LIN {X 0,Y 318.521,Z 646.616,A -85,B 0,C 180,E1 12916.819,E2 12916.819} C_VEL
LIN {X 0,Y 314.877,Z 667.549,A -85,B 0,C 180,E1 12915.793,E2 12915.793} C_VEL
LIN {X 0,Y 310.481,Z 687.705,A -85,B 0,C 180,E1 12914.459,E2 12914.459} C_VEL
LIN {X 0,Y 305.511,Z 707.389,A -85,B 0,C 180,E1 12912.755,E2 12912.755} C_VEL
LIN {X 0,Y 300.341,Z 725.782,A -85,B 0,C 180,E1 12910.729,E2 12910.729} C_VEL
LIN {X 0,Y 295.179,Z 742.727,A -85,B 0,C 180,E1 12908.414,E2 12908.414} C_VEL
LIN {X 0,Y 290.123,Z 758.694,A -85,B 0,C 180,E1 12905.742,E2 12905.742} C_VEL
LIN {X 0,Y 285.541,Z 773.07,A -85,B 0,C 180,E1 12902.819,E2 12902.819} C_VEL
LIN {X 0,Y 281.238,Z 787.006,A -85,B 0,C 180,E1 12899.38,E2 12899.38} C_VEL
LIN {X 0,Y 277.714,Z 799.537,A -85,B 0,C 180,E1 12895.596,E2 12895.596} C_VEL
LIN {X 0,Y 275.265,Z 809.934,A -85,B 0,C 180,E1 12891.746,E2 12891.746} C_VEL
LIN {X 0,Y 273.777,Z 818.455,A -85,B 0,C 180,E1 12887.864,E2 12887.864} C_VEL
LIN {X 0,Y 273.13,Z 825.558,A -85,B 0,C 180,E1 12883.765,E2 12883.765} C_VEL
LIN {X 0,Y 273.196,Z 830.779,A -85,B 0,C 180,E1 12879.692,E2 12879.692} C_VEL
LIN {X 0,Y 273.612,Z 834.096,A -85,B 0,C 180,E1 12875.873,E2 12875.873} C_VEL
LIN {X 0,Y 273.979,Z 835.824,A -85,B 0,C 180,E1 12872.301,E2 12872.301} C_VEL
LIN {X 0,Y 274.057,Z 836.01,A -85,B 0,C 180,E1 12868.955,E2 12868.955} C_VEL
LIN {X 0,Y 273.763,Z 834.896,A -85,B 0,C 180,E1 12865.391,E2 12865.391} C_VEL
LIN {X 0,Y 273.337,Z 832.235,A -85,B 0,C 180,E1 12861.798,E2 12861.798} C_VEL
LIN {X 0,Y 273.084,Z 827.633,A -85,B 0,C 180,E1 12857.74,E2 12857.74} C_VEL
LIN {X 0,Y 273.452,Z 821.244,A -85,B 0,C 180,E1 12853.648,E2 12853.648} C_VEL
LIN {X 0,Y 274.661,Z 812.965,A -85,B 0,C 180,E1 12849.546,E2 12849.546} C_VEL
LIN {X 0,Y 276.918,Z 802.631,A -85,B 0,C 180,E1 12845.467,E2 12845.467} C_VEL
LIN {X 0,Y 280.149,Z 790.716,A -85,B 0,C 180,E1 12841.662,E2 12841.662} C_VEL
LIN {X 0,Y 284.213,Z 777.257,A -85,B 0,C 180,E1 12838.151,E2 12838.151} C_VEL
LIN {X 0,Y 288.798,Z 762.744,A -85,B 0,C 180,E1 12835.043,E2 12835.043} C_VEL
LIN {X 0,Y 293.673,Z 747.357,A -85,B 0,C 180,E1 12832.329,E2 12832.329} C_VEL
LIN {X 0,Y 298.826,Z 730.575,A -85,B 0,C 180,E1 12829.903,E2 12829.903} C_VEL
LIN {X 0,Y 304.127,Z 712.146,A -85,B 0,C 180,E1 12827.755,E2 12827.755} C_VEL
LIN {X 0,Y 309.042,Z 693.226,A -85,B 0,C 180,E1 12826.004,E2 12826.004} C_VEL
LIN {X 0,Y 313.618,Z 673.067,A -85,B 0,C 180,E1 12824.559,E2 12824.559} C_VEL
LIN {X 0,Y 317.514,Z 652.33,A -85,B 0,C 180,E1 12823.454,E2 12823.454} C_VEL
LIN {X 0,Y 320.333,Z 631.352,A -85,B 0,C 180,E1 12822.639,E2 12822.639} C_VEL
LIN {X 0,Y 322.11,Z 608.021,A -85,B 0,C 180,E1 12822.015,E2 12822.015} C_VEL
LIN {X 0,Y 331.889,Z 436.421,A -85,B 0,C 180,E1 12818.133,E2 12818.133} C_VEL
LIN {X 0,Y 331.118,Z 424.68,A -85,B 0,C 180,E1 12817.587,E2 12817.587} C_VEL
LIN {X 0,Y 322.829,Z 409.225,A -85,B 0,C 180,E1 12815.31,E2 12815.31} C_VEL
LIN {X 0,Y 314.205,Z 394.789,A -85,B 0,C 180,E1 12812.749,E2 12812.749} C_VEL
LIN {X 0,Y 306.355,Z 382.678,A -85,B 0,C 180,E1 12810.173,E2 12810.173} C_VEL
LIN {X 0,Y 298.711,Z 371.628,A -85,B 0,C 180,E1 12807.349,E2 12807.349} C_VEL
LIN {X 0,Y 294.503,Z 363.438,A -85,B 0,C 180,E1 12804.255,E2 12804.255} C_VEL
LIN {X 0,Y 291.847,Z 358.564,A -85,B 0,C 180,E1 12802.139,E2 12802.139} C_VEL
LIN {X 0,Y 289.754,Z 354.487,A -85,B 0,C 180,E1 12800.186,E2 12800.186} C_VEL
LIN {X 0,Y 287.159,Z 349.76,A -85,B 0,C 180,E1 12797.633,E2 12797.633} C_VEL
LIN {X 0,Y 284.83,Z 345.563,A -85,B 0,C 180,E1 12795.056,E2 12795.056} C_VEL
LIN {X 0,Y 281.786,Z 340.679,A -85,B 0,C 180,E1 12791.253,E2 12791.253} C_VEL
LIN {X 0,Y 281.192,Z 339.431,A -85,B 0,C 180,E1 12790.241,E2 12790.241} C_VEL
LIN {X 0,Y 277.823,Z 333.98,A -85,B 0,C 180,E1 12783.507,E2 12783.507} C_VEL
LIN {X 0,Y 276.215,Z 332.418,A -85,B 0,C 180,E1 12777.505,E2 12777.505} C_VEL
LIN {X 0,Y 276.38,Z 332.578,A -85,B 0,C 180,E1 12772.098,E2 12772.098} C_VEL
LIN {X 0,Y 277.952,Z 334.225,A -85,B 0,C 180,E1 12766.901,E2 12766.901} C_VEL
LIN {X 0,Y 281.193,Z 339.671,A -85,B 0,C 180,E1 12760.257,E2 12760.257} C_VEL
LIN {X 0,Y 283.306,Z 343.892,A -85,B 0,C 180,E1 12756.936,E2 12756.936} C_VEL
LIN {X 0,Y 284.176,Z 345.216,A -85,B 0,C 180,E1 12755.911,E2 12755.911} C_VEL
LIN {X 0,Y 286.766,Z 350.132,A -85,B 0,C 180,E1 12752.757,E2 12752.757} C_VEL
LIN {X 0,Y 289.262,Z 355.103,A -85,B 0,C 180,E1 12750.034,E2 12750.034} C_VEL
LIN {X 0,Y 295.268,Z 362.715,A -85,B 0,C 180,E1 12747.366,E2 12747.366} C_VEL
LIN {X 0,Y 303.925,Z 373.809,A -85,B 0,C 180,E1 12744.097,E2 12744.097} C_VEL
LIN {X 0,Y 313.853,Z 387.94,A -85,B 0,C 180,E1 12740.833,E2 12740.833} C_VEL
LIN {X 0,Y 323.057,Z 402.598,A -85,B 0,C 180,E1 12738.136,E2 12738.136} C_VEL
LIN {X 0,Y 331.436,Z 417.301,A -85,B 0,C 180,E1 12735.892,E2 12735.892} C_VEL
LIN {X 0,Y 324.029,Z 570.746,A -85,B 0,C 180,E1 12732.693,E2 12732.693} C_VEL
LIN {X 0,Y 322.622,Z 590.161,A -85,B 0,C 180,E1 12732.013,E2 12732.013} C_VEL
LIN {X 0,Y 320.358,Z 608.777,A -85,B 0,C 180,E1 12731.069,E2 12731.069} C_VEL
LIN {X 0,Y 317.4,Z 626.429,A -85,B 0,C 180,E1 12729.869,E2 12729.869} C_VEL
LIN {X 0,Y 313.615,Z 644.125,A -85,B 0,C 180,E1 12728.322,E2 12728.322} C_VEL
LIN {X 0,Y 309.308,Z 660.695,A -85,B 0,C 180,E1 12726.497,E2 12726.497} C_VEL
LIN {X 0,Y 304.53,Z 676.538,A -85,B 0,C 180,E1 12724.313,E2 12724.313} C_VEL
LIN {X 0,Y 299.564,Z 691.068,A -85,B 0,C 180,E1 12721.826,E2 12721.826} C_VEL
LIN {X 0,Y 294.635,Z 704.227,A -85,B 0,C 180,E1 12719.03,E2 12719.03} C_VEL
LIN {X 0,Y 289.962,Z 715.814,A -85,B 0,C 180,E1 12715.971,E2 12715.971} C_VEL
LIN {X 0,Y 285.729,Z 725.888,A -85,B 0,C 180,E1 12712.638,E2 12712.638} C_VEL
LIN {X 0,Y 282.058,Z 734.454,A -85,B 0,C 180,E1 12709.033,E2 12709.033} C_VEL
LIN {X 0,Y 279.071,Z 741.482,A -85,B 0,C 180,E1 12705.161,E2 12705.161} C_VEL
LIN {X 0,Y 276.972,Z 746.671,A -85,B 0,C 180,E1 12701.241,E2 12701.241} C_VEL
LIN {X 0,Y 275.562,Z 750.342,A -85,B 0,C 180,E1 12697.086,E2 12697.086} C_VEL
LIN {X 0,Y 274.872,Z 752.306,A -85,B 0,C 180,E1 12692.919,E2 12692.919} C_VEL
LIN {X 0,Y 274.762,Z 752.649,A -85,B 0,C 180,E1 12688.749,E2 12688.749} C_VEL
LIN {X 0,Y 275.198,Z 751.384,A -85,B 0,C 180,E1 12684.572,E2 12684.572} C_VEL
LIN {X 0,Y 276.288,Z 748.463,A -85,B 0,C 180,E1 12680.418,E2 12680.418} C_VEL
LIN {X 0,Y 278.158,Z 743.76,A -85,B 0,C 180,E1 12676.277,E2 12676.277} C_VEL
LIN {X 0,Y 280.792,Z 737.489,A -85,B 0,C 180,E1 12672.382,E2 12672.382} C_VEL
LIN {X 0,Y 284.139,Z 729.734,A -85,B 0,C 180,E1 12668.75,E2 12668.75} C_VEL
LIN {X 0,Y 288.037,Z 720.554,A -85,B 0,C 180,E1 12665.384,E2 12665.384} C_VEL
LIN {X 0,Y 292.411,Z 709.978,A -85,B 0,C 180,E1 12662.289,E2 12662.289} C_VEL
LIN {X 0,Y 297.09,Z 698.005,A -85,B 0,C 180,E1 12659.458,E2 12659.458} C_VEL
LIN {X 0,Y 302.111,Z 684.038,A -85,B 0,C 180,E1 12656.789,E2 12656.789} C_VEL
LIN {X 0,Y 307.017,Z 668.867,A -85,B 0,C 180,E1 12654.458,E2 12654.458} C_VEL
LIN {X 0,Y 311.62,Z 652.509,A -85,B 0,C 180,E1 12652.438,E2 12652.438} C_VEL
LIN {X 0,Y 315.588,Z 635.868,A -85,B 0,C 180,E1 12650.799,E2 12650.799} C_VEL
LIN {X 0,Y 318.977,Z 618.266,A -85,B 0,C 180,E1 12649.428,E2 12649.428} C_VEL
LIN {X 0,Y 321.711,Z 599.435,A -85,B 0,C 180,E1 12648.312,E2 12648.312} C_VEL
LIN {X 0,Y 323.578,Z 579.916,A -85,B 0,C 180,E1 12647.482,E2 12647.482} C_VEL
LIN {X 0,Y 324.743,Z 555.923,A -85,B 0,C 180,E1 12646.846,E2 12646.846} C_VEL
LIN {X 0,Y 325.912,Z 530.757,A -85,B 0,C 180,E1 12646.323,E2 12646.323} C_VEL
LIN {X 0,Y 325.604,Z 523.168,A -85,B 0,C 180,E1 12646.04,E2 12646.04} C_VEL
LIN {X 0,Y 322.384,Z 503.34,A -85,B 0,C 180,E1 12644.815,E2 12644.815} C_VEL
LIN {X 0,Y 322.193,Z 496.818,A -85,B 0,C 180,E1 12644.576,E2 12644.576} C_VEL
LIN {X 0,Y 326.056,Z 420.531,A -85,B 0,C 180,E1 12642.97,E2 12642.97} C_VEL
LIN {X 0,Y 317.729,Z 405.913,A -85,B 0,C 180,E1 12640.619,E2 12640.619} C_VEL
LIN {X 0,Y 309.549,Z 392.937,A -85,B 0,C 180,E1 12638.093,E2 12638.093} C_VEL
LIN {X 0,Y 300.513,Z 379.839,A -85,B 0,C 180,E1 12634.968,E2 12634.968} C_VEL
LIN {X 0,Y 291.185,Z 367.626,A -85,B 0,C 180,E1 12631.232,E2 12631.232} C_VEL
LIN {X 0,Y 285.424,Z 360.648,A -85,B 0,C 180,E1 12628.566,E2 12628.566} C_VEL
LIN {X 0,Y 281.908,Z 356.155,A -85,B 0,C 180,E1 12626.651,E2 12626.651} C_VEL
LIN {X 0,Y 279.002,Z 350.696,A -85,B 0,C 180,E1 12622.93,E2 12622.93} C_VEL
LIN {X 0,Y 276.761,Z 346.463,A -85,B 0,C 180,E1 12619.413,E2 12619.413} C_VEL
LIN {X 0,Y 273.571,Z 340.764,A -85,B 0,C 180,E1 12612.025,E2 12612.025} C_VEL
LIN {X 0,Y 272.202,Z 339.441,A -85,B 0,C 180,E1 12606.327,E2 12606.327} C_VEL
LIN {X 0,Y 272.456,Z 339.661,A -85,B 0,C 180,E1 12601.262,E2 12601.262} C_VEL
LIN {X 0,Y 273.881,Z 341.096,A -85,B 0,C 180,E1 12596.442,E2 12596.442} C_VEL
LIN {X 0,Y 277.267,Z 346.64,A -85,B 0,C 180,E1 12589.613,E2 12589.613} C_VEL
LIN {X 0,Y 279.445,Z 350.884,A -85,B 0,C 180,E1 12586.341,E2 12586.341} C_VEL
LIN {X 0,Y 280.36,Z 352.123,A -85,B 0,C 180,E1 12585.333,E2 12585.333} C_VEL
LIN {X 0,Y 282.589,Z 356.255,A -85,B 0,C 180,E1 12582.71,E2 12582.71} C_VEL
LIN {X 0,Y 285.907,Z 362.472,A -85,B 0,C 180,E1 12579.317,E2 12579.317} C_VEL
LIN {X 0,Y 288.869,Z 368.159,A -85,B 0,C 180,E1 12576.76,E2 12576.76} C_VEL
LIN {X 0,Y 290.863,Z 371.534,A -85,B 0,C 180,E1 12575.422,E2 12575.422} C_VEL
LIN {X 0,Y 298.308,Z 382.017,A -85,B 0,C 180,E1 12572.341,E2 12572.341} C_VEL
LIN {X 0,Y 306.047,Z 393.465,A -85,B 0,C 180,E1 12569.523,E2 12569.523} C_VEL
LIN {X 0,Y 314.219,Z 406.761,A -85,B 0,C 180,E1 12566.845,E2 12566.845} C_VEL
LIN {X 0,Y 323.159,Z 422.766,A -85,B 0,C 180,E1 12564.186,E2 12564.186} C_VEL
LIN {X 0,Y 326.324,Z 429.459,A -85,B 0,C 180,E1 12563.27,E2 12563.27} C_VEL
LIN {X 0,Y 326.603,Z 440.209,A -85,B 0,C 180,E1 12562.833,E2 12562.833} C_VEL
LIN {X 0,Y 315.481,Z 623.904,A -85,B 0,C 180,E1 12558.626,E2 12558.626} C_VEL
LIN {X 0,Y 312.841,Z 645.686,A -85,B 0,C 180,E1 12557.856,E2 12557.856} C_VEL
LIN {X 0,Y 309.118,Z 666.476,A -85,B 0,C 180,E1 12556.834,E2 12556.834} C_VEL
LIN {X 0,Y 304.704,Z 686.073,A -85,B 0,C 180,E1 12555.536,E2 12555.536} C_VEL
LIN {X 0,Y 299.76,Z 704.977,A -85,B 0,C 180,E1 12553.907,E2 12553.907} C_VEL
LIN {X 0,Y 294.582,Z 722.809,A -85,B 0,C 180,E1 12551.961,E2 12551.961} C_VEL
LIN {X 0,Y 289.168,Z 739.981,A -85,B 0,C 180,E1 12549.637,E2 12549.637} C_VEL
LIN {X 0,Y 283.936,Z 755.721,A -85,B 0,C 180,E1 12547.024,E2 12547.024} C_VEL
LIN {X 0,Y 278.946,Z 770.642,A -85,B 0,C 180,E1 12543.997,E2 12543.997} C_VEL
LIN {X 0,Y 274.482,Z 784.174,A -85,B 0,C 180,E1 12540.661,E2 12540.661} C_VEL
LIN {X 0,Y 270.765,Z 796.349,A -85,B 0,C 180,E1 12537.013,E2 12537.013} C_VEL
LIN {X 0,Y 267.921,Z 807.109,A -85,B 0,C 180,E1 12533.069,E2 12533.069} C_VEL
LIN {X 0,Y 266.005,Z 816.654,A -85,B 0,C 180,E1 12528.7,E2 12528.7} C_VEL
LIN {X 0,Y 265.206,Z 823.96,A -85,B 0,C 180,E1 12524.408,E2 12524.408} C_VEL
LIN {X 0,Y 265.204,Z 829.303,A -85,B 0,C 180,E1 12520.206,E2 12520.206} C_VEL
LIN {X 0,Y 265.626,Z 832.742,A -85,B 0,C 180,E1 12516.267,E2 12516.267} C_VEL
LIN {X 0,Y 266.028,Z 834.465,A -85,B 0,C 180,E1 12512.8,E2 12512.8} C_VEL
LIN {X 0,Y 266.157,Z 834.862,A -85,B 0,C 180,E1 12509.354,E2 12509.354} C_VEL
LIN {X 0,Y 265.922,Z 834.045,A -85,B 0,C 180,E1 12506.119,E2 12506.119} C_VEL
LIN {X 0,Y 265.435,Z 831.58,A -85,B 0,C 180,E1 12502.206,E2 12502.206} C_VEL
LIN {X 0,Y 265.12,Z 827.563,A -85,B 0,C 180,E1 12498.25,E2 12498.25} C_VEL
LIN {X 0,Y 265.396,Z 821.493,A -85,B 0,C 180,E1 12494.037,E2 12494.037} C_VEL
LIN {X 0,Y 266.529,Z 813.563,A -85,B 0,C 180,E1 12489.811,E2 12489.811} C_VEL
LIN {X 0,Y 268.637,Z 804.049,A -85,B 0,C 180,E1 12485.766,E2 12485.766} C_VEL
LIN {X 0,Y 271.757,Z 792.882,A -85,B 0,C 180,E1 12481.905,E2 12481.905} C_VEL
LIN {X 0,Y 275.768,Z 780.085,A -85,B 0,C 180,E1 12478.284,E2 12478.284} C_VEL
LIN {X 0,Y 280.514,Z 765.839,A -85,B 0,C 180,E1 12474.981,E2 12474.981} C_VEL
LIN {X 0,Y 285.698,Z 750.379,A -85,B 0,C 180,E1 12472.046,E2 12472.046} C_VEL
LIN {X 0,Y 291.038,Z 734.033,A -85,B 0,C 180,E1 12469.512,E2 12469.512} C_VEL
LIN {X 0,Y 296.423,Z 716.509,A -85,B 0,C 180,E1 12467.315,E2 12467.315} C_VEL
LIN {X 0,Y 301.818,Z 697.169,A -85,B 0,C 180,E1 12465.389,E2 12465.389} C_VEL
LIN {X 0,Y 306.581,Z 677.71,A -85,B 0,C 180,E1 12463.885,E2 12463.885} C_VEL
LIN {X 0,Y 310.665,Z 657.913,A -85,B 0,C 180,E1 12462.727,E2 12462.727} C_VEL
LIN {X 0,Y 313.859,Z 637.577,A -85,B 0,C 180,E1 12461.847,E2 12461.847} C_VEL
LIN {X 0,Y 315.922,Z 616.704,A -85,B 0,C 180,E1 12461.203,E2 12461.203} C_VEL
LIN {X 0,Y 326.575,Z 437.654,A -85,B 0,C 180,E1 12457.112,E2 12457.112} C_VEL
LIN {X 0,Y 326.002,Z 428.555,A -85,B 0,C 180,E1 12456.677,E2 12456.677} C_VEL
LIN {X 0,Y 317.855,Z 413.201,A -85,B 0,C 180,E1 12454.323,E2 12454.323} C_VEL
LIN {X 0,Y 308.899,Z 398.062,A -85,B 0,C 180,E1 12451.517,E2 12451.517} C_VEL
LIN {X 0,Y 300.403,Z 384.981,A -85,B 0,C 180,E1 12448.53,E2 12448.53} C_VEL
LIN {X 0,Y 292.847,Z 374.376,A -85,B 0,C 180,E1 12445.534,E2 12445.534} C_VEL
LIN {X 0,Y 290.063,Z 370.213,A -85,B 0,C 180,E1 12444.217,E2 12444.217} C_VEL
LIN {X 0,Y 286.914,Z 364.504,A -85,B 0,C 180,E1 12441.678,E2 12441.678} C_VEL
LIN {X 0,Y 284.984,Z 360.764,A -85,B 0,C 180,E1 12439.896,E2 12439.896} C_VEL
LIN {X 0,Y 282.411,Z 356.076,A -85,B 0,C 180,E1 12437.301,E2 12437.301} C_VEL
LIN {X 0,Y 279.905,Z 351.338,A -85,B 0,C 180,E1 12434.269,E2 12434.269} C_VEL
LIN {X 0,Y 277.516,Z 347.594,A -85,B 0,C 180,E1 12431.218,E2 12431.218} C_VEL
LIN {X 0,Y 276.813,Z 346.091,A -85,B 0,C 180,E1 12429.984,E2 12429.984} C_VEL
LIN {X 0,Y 273.63,Z 340.766,A -85,B 0,C 180,E1 12423.351,E2 12423.351} C_VEL
LIN {X 0,Y 272.02,Z 339.216,A -85,B 0,C 180,E1 12417.261,E2 12417.261} C_VEL
LIN {X 0,Y 272.217,Z 339.429,A -85,B 0,C 180,E1 12411.976,E2 12411.976} C_VEL
LIN {X 0,Y 273.675,Z 341.008,A -85,B 0,C 180,E1 12406.908,E2 12406.908} C_VEL
LIN {X 0,Y 276.735,Z 346.396,A -85,B 0,C 180,E1 12400.365,E2 12400.365} C_VEL
LIN {X 0,Y 278.871,Z 350.546,A -85,B 0,C 180,E1 12396.995,E2 12396.995} C_VEL
LIN {X 0,Y 279.602,Z 351.984,A -85,B 0,C 180,E1 12395.941,E2 12395.941} C_VEL
LIN {X 0,Y 282.03,Z 356.488,A -85,B 0,C 180,E1 12393.012,E2 12393.012} C_VEL
LIN {X 0,Y 285.873,Z 361.055,A -85,B 0,C 180,E1 12391.026,E2 12391.026} C_VEL
LIN {X 0,Y 292.839,Z 369.89,A -85,B 0,C 180,E1 12387.873,E2 12387.873} C_VEL
LIN {X 0,Y 300.999,Z 380.593,A -85,B 0,C 180,E1 12384.69,E2 12384.69} C_VEL
LIN {X 0,Y 310.626,Z 394.567,A -85,B 0,C 180,E1 12381.416,E2 12381.416} C_VEL
LIN {X 0,Y 319.403,Z 408.86,A -85,B 0,C 180,E1 12378.75,E2 12378.75} C_VEL
LIN {X 0,Y 326.078,Z 420.895,A -85,B 0,C 180,E1 12376.879,E2 12376.879} C_VEL
LIN {X 0,Y 318.463,Z 571.358,A -85,B 0,C 180,E1 12373.711,E2 12373.711} C_VEL
LIN {X 0,Y 316.99,Z 590.894,A -85,B 0,C 180,E1 12373.022,E2 12373.022} C_VEL
LIN {X 0,Y 314.593,Z 609.838,A -85,B 0,C 180,E1 12372.052,E2 12372.052} C_VEL
LIN {X 0,Y 311.344,Z 628.339,A -85,B 0,C 180,E1 12370.771,E2 12370.771} C_VEL
LIN {X 0,Y 307.479,Z 645.583,A -85,B 0,C 180,E1 12369.232,E2 12369.232} C_VEL
LIN {X 0,Y 303.009,Z 662.069,A -85,B 0,C 180,E1 12367.383,E2 12367.383} C_VEL
LIN {X 0,Y 298.164,Z 677.501,A -85,B 0,C 180,E1 12365.223,E2 12365.223} C_VEL
LIN {X 0,Y 293.241,Z 691.381,A -85,B 0,C 180,E1 12362.828,E2 12362.828} C_VEL
LIN {X 0,Y 288.068,Z 704.681,A -85,B 0,C 180,E1 12359.987,E2 12359.987} C_VEL
LIN {X 0,Y 283.147,Z 716.394,A -85,B 0,C 180,E1 12356.871,E2 12356.871} C_VEL
LIN {X 0,Y 278.666,Z 726.58,A -85,B 0,C 180,E1 12353.469,E2 12353.469} C_VEL
LIN {X 0,Y 274.765,Z 735.247,A -85,B 0,C 180,E1 12349.78,E2 12349.78} C_VEL
LIN {X 0,Y 271.565,Z 742.37,A -85,B 0,C 180,E1 12345.81,E2 12345.81} C_VEL
LIN {X 0,Y 269.2,Z 747.878,A -85,B 0,C 180,E1 12341.57,E2 12341.57} C_VEL
LIN {X 0,Y 267.705,Z 751.546,A -85,B 0,C 180,E1 12337.295,E2 12337.295} C_VEL
LIN {X 0,Y 266.971,Z 753.508,A -85,B 0,C 180,E1 12333.006,E2 12333.006} C_VEL
LIN {X 0,Y 266.854,Z 753.851,A -85,B 0,C 180,E1 12328.712,E2 12328.712} C_VEL
LIN {X 0,Y 267.317,Z 752.59,A -85,B 0,C 180,E1 12324.419,E2 12324.419} C_VEL
LIN {X 0,Y 268.477,Z 749.667,A -85,B 0,C 180,E1 12320.136,E2 12320.136} C_VEL
LIN {X 0,Y 270.459,Z 744.967,A -85,B 0,C 180,E1 12315.878,E2 12315.878} C_VEL
LIN {X 0,Y 273.239,Z 738.7,A -85,B 0,C 180,E1 12311.879,E2 12311.879} C_VEL
LIN {X 0,Y 276.759,Z 730.951,A -85,B 0,C 180,E1 12308.155,E2 12308.155} C_VEL
LIN {X 0,Y 280.849,Z 721.782,A -85,B 0,C 180,E1 12304.71,E2 12304.71} C_VEL
LIN {X 0,Y 285.424,Z 711.219,A -85,B 0,C 180,E1 12301.549,E2 12301.549} C_VEL
LIN {X 0,Y 290.65,Z 698.387,A -85,B 0,C 180,E1 12298.475,E2 12298.475} C_VEL
LIN {X 0,Y 295.722,Z 684.799,A -85,B 0,C 180,E1 12295.858,E2 12295.858} C_VEL
LIN {X 0,Y 300.837,Z 669.56,A -85,B 0,C 180,E1 12293.494,E2 12293.494} C_VEL
LIN {X 0,Y 305.413,Z 653.91,A -85,B 0,C 180,E1 12291.538,E2 12291.538} C_VEL
LIN {X 0,Y 309.751,Z 636.388,A -85,B 0,C 180,E1 12289.792,E2 12289.792} C_VEL
LIN {X 0,Y 313.272,Z 618.661,A -85,B 0,C 180,E1 12288.406,E2 12288.406} C_VEL
LIN {X 0,Y 316.124,Z 599.539,A -85,B 0,C 180,E1 12287.272,E2 12287.272} C_VEL
LIN {X 0,Y 318.041,Z 579.955,A -85,B 0,C 180,E1 12286.444,E2 12286.444} C_VEL
LIN {X 0,Y 319.275,Z 555.252,A -85,B 0,C 180,E1 12285.793,E2 12285.793} C_VEL
LIN {X 0,Y 322.193,Z 496.818,A -85,B 0,C 180,E1 12284.576,E2 12284.576} C_VEL
LIN {X 0,Y 321.9,Z 489.233,A -85,B 0,C 180,E1 12284.281,E2 12284.281} C_VEL
LIN {X 0,Y 318.898,Z 469.415,A -85,B 0,C 180,E1 12283.022,E2 12283.022} C_VEL
LIN {X 0,Y 318.781,Z 462.892,A -85,B 0,C 180,E1 12282.784,E2 12282.784} C_VEL
LIN {X 0,Y 320.861,Z 424.086,A -85,B 0,C 180,E1 12281.958,E2 12281.958} C_VEL
LIN {X 0,Y 312.608,Z 409.503,A -85,B 0,C 180,E1 12279.501,E2 12279.501} C_VEL
LIN {X 0,Y 303.827,Z 395.623,A -85,B 0,C 180,E1 12276.618,E2 12276.618} C_VEL
LIN {X 0,Y 295.497,Z 383.738,A -85,B 0,C 180,E1 12273.531,E2 12273.531} C_VEL
LIN {X 0,Y 287.709,Z 373.406,A -85,B 0,C 180,E1 12270.202,E2 12270.202} C_VEL
LIN {X 0,Y 282.994,Z 367.663,A -85,B 0,C 180,E1 12267.914,E2 12267.914} C_VEL
LIN {X 0,Y 278.943,Z 362.711,A -85,B 0,C 180,E1 12265.704,E2 12265.704} C_VEL
LIN {X 0,Y 275.103,Z 358.176,A -85,B 0,C 180,E1 12263.339,E2 12263.339} C_VEL
LIN {X 0,Y 274.001,Z 356.757,A -85,B 0,C 180,E1 12262.304,E2 12262.304} C_VEL
LIN {X 0,Y 272.017,Z 352.491,A -85,B 0,C 180,E1 12258.651,E2 12258.651} C_VEL
LIN {X 0,Y 269.226,Z 347.427,A -85,B 0,C 180,E1 12251.787,E2 12251.787} C_VEL
LIN {X 0,Y 268.004,Z 346.218,A -85,B 0,C 180,E1 12245.782,E2 12245.782} C_VEL
LIN {X 0,Y 268.413,Z 346.646,A -85,B 0,C 180,E1 12240.641,E2 12240.641} C_VEL
LIN {X 0,Y 269.761,Z 347.998,A -85,B 0,C 180,E1 12236.388,E2 12236.388} C_VEL
LIN {X 0,Y 272.967,Z 353.552,A -85,B 0,C 180,E1 12229.661,E2 12229.661} C_VEL
LIN {X 0,Y 275.149,Z 357.655,A -85,B 0,C 180,E1 12226.338,E2 12226.338} C_VEL
LIN {X 0,Y 275.934,Z 359.08,A -85,B 0,C 180,E1 12225.307,E2 12225.307} C_VEL
LIN {X 0,Y 278.607,Z 363.943,A -85,B 0,C 180,E1 12222.239,E2 12222.239} C_VEL
LIN {X 0,Y 281.536,Z 369.341,A -85,B 0,C 180,E1 12219.416,E2 12219.416} C_VEL
LIN {X 0,Y 288.409,Z 378.688,A -85,B 0,C 180,E1 12215.962,E2 12215.962} C_VEL
LIN {X 0,Y 295.489,Z 388.867,A -85,B 0,C 180,E1 12212.928,E2 12212.928} C_VEL
LIN {X 0,Y 302.956,Z 400.202,A -85,B 0,C 180,E1 12210.109,E2 12210.109} C_VEL
LIN {X 0,Y 310.665,Z 413.045,A -85,B 0,C 180,E1 12207.488,E2 12207.488} C_VEL
LIN {X 0,Y 319.096,Z 428.488,A -85,B 0,C 180,E1 12204.875,E2 12204.875} C_VEL
LIN {X 0,Y 321.258,Z 433.222,A -85,B 0,C 180,E1 12204.217,E2 12204.217} C_VEL
LIN {X 0,Y 321.382,Z 441.415,A -85,B 0,C 180,E1 12203.892,E2 12203.892} C_VEL
LIN {X 0,Y 309.98,Z 622.999,A -85,B 0,C 180,E1 12199.705,E2 12199.705} C_VEL
LIN {X 0,Y 307.28,Z 644.682,A -85,B 0,C 180,E1 12198.935,E2 12198.935} C_VEL
LIN {X 0,Y 303.47,Z 665.37,A -85,B 0,C 180,E1 12197.916,E2 12197.916} C_VEL
LIN {X 0,Y 298.765,Z 685.59,A -85,B 0,C 180,E1 12196.569,E2 12196.569} C_VEL
LIN {X 0,Y 293.432,Z 705.157,A -85,B 0,C 180,E1 12194.856,E2 12194.856} C_VEL
LIN {X 0,Y 287.796,Z 723.659,A -85,B 0,C 180,E1 12192.78,E2 12192.78} C_VEL
LIN {X 0,Y 282.026,Z 741.029,A -85,B 0,C 180,E1 12190.339,E2 12190.339} C_VEL
LIN {X 0,Y 276.407,Z 757.054,A -85,B 0,C 180,E1 12187.554,E2 12187.554} C_VEL
LIN {X 0,Y 271.431,Z 771.124,A -85,B 0,C 180,E1 12184.56,E2 12184.56} C_VEL
LIN {X 0,Y 266.554,Z 785.146,A -85,B 0,C 180,E1 12180.923,E2 12180.923} C_VEL
LIN {X 0,Y 262.573,Z 797.58,A -85,B 0,C 180,E1 12176.945,E2 12176.945} C_VEL
LIN {X 0,Y 259.636,Z 808.401,A -85,B 0,C 180,E1 12172.649,E2 12172.649} C_VEL
LIN {X 0,Y 257.828,Z 817.539,A -85,B 0,C 180,E1 12168.073,E2 12168.073} C_VEL
LIN {X 0,Y 257.177,Z 824.425,A -85,B 0,C 180,E1 12163.603,E2 12163.603} C_VEL
LIN {X 0,Y 257.326,Z 829.321,A -85,B 0,C 180,E1 12159.275,E2 12159.275} C_VEL
LIN {X 0,Y 257.81,Z 832.213,A -85,B 0,C 180,E1 12155.341,E2 12155.341} C_VEL
LIN {X 0,Y 258.192,Z 833.52,A -85,B 0,C 180,E1 12151.775,E2 12151.775} C_VEL
LIN {X 0,Y 258.221,Z 833.577,A -85,B 0,C 180,E1 12148.669,E2 12148.669} C_VEL
LIN {X 0,Y 257.873,Z 832.472,A -85,B 0,C 180,E1 12145.107,E2 12145.107} C_VEL
LIN {X 0,Y 257.392,Z 829.782,A -85,B 0,C 180,E1 12141.286,E2 12141.286} C_VEL
LIN {X 0,Y 257.157,Z 825.142,A -85,B 0,C 180,E1 12136.967,E2 12136.967} C_VEL
LIN {X 0,Y 257.649,Z 818.824,A -85,B 0,C 180,E1 12132.678,E2 12132.678} C_VEL
LIN {X 0,Y 259.172,Z 810.403,A -85,B 0,C 180,E1 12128.263,E2 12128.263} C_VEL
LIN {X 0,Y 261.847,Z 800.038,A -85,B 0,C 180,E1 12123.953,E2 12123.953} C_VEL
LIN {X 0,Y 265.565,Z 788.098,A -85,B 0,C 180,E1 12119.951,E2 12119.951} C_VEL
LIN {X 0,Y 270.179,Z 774.612,A -85,B 0,C 180,E1 12116.283,E2 12116.283} C_VEL
LIN {X 0,Y 275.675,Z 759.061,A -85,B 0,C 180,E1 12112.852,E2 12112.852} C_VEL
LIN {X 0,Y 281.544,Z 742.29,A -85,B 0,C 180,E1 12109.876,E2 12109.876} C_VEL
LIN {X 0,Y 287.32,Z 724.95,A -85,B 0,C 180,E1 12107.403,E2 12107.403} C_VEL
LIN {X 0,Y 292.908,Z 706.657,A -85,B 0,C 180,E1 12105.318,E2 12105.318} C_VEL
LIN {X 0,Y 298.194,Z 687.393,A -85,B 0,C 180,E1 12103.595,E2 12103.595} C_VEL
LIN {X 0,Y 302.716,Z 668.307,A -85,B 0,C 180,E1 12102.282,E2 12102.282} C_VEL
LIN {X 0,Y 306.579,Z 648.218,A -85,B 0,C 180,E1 12101.243,E2 12101.243} C_VEL
LIN {X 0,Y 309.402,Z 627.413,A -85,B 0,C 180,E1 12100.455,E2 12100.455} C_VEL
LIN {X 0,Y 311.513,Z 598.823,A -85,B 0,C 180,E1 12099.718,E2 12099.718} C_VEL
LIN {X 0,Y 321.355,Z 438.503,A -85,B 0,C 180,E1 12096.039,E2 12096.039} C_VEL
LIN {X 0,Y 320.98,Z 432.39,A -85,B 0,C 180,E1 12095.737,E2 12095.737} C_VEL
LIN {X 0,Y 312.401,Z 416.174,A -85,B 0,C 180,E1 12093.127,E2 12093.127} C_VEL
LIN {X 0,Y 303.613,Z 401.378,A -85,B 0,C 180,E1 12090.201,E2 12090.201} C_VEL
LIN {X 0,Y 295.853,Z 389.496,A -85,B 0,C 180,E1 12087.308,E2 12087.308} C_VEL
LIN {X 0,Y 289.927,Z 380.953,A -85,B 0,C 180,E1 12084.826,E2 12084.826} C_VEL
LIN {X 0,Y 286.251,Z 375.895,A -85,B 0,C 180,E1 12083.138,E2 12083.138} C_VEL
LIN {X 0,Y 281.219,Z 368.69,A -85,B 0,C 180,E1 12080.391,E2 12080.391} C_VEL
LIN {X 0,Y 277.967,Z 362.69,A -85,B 0,C 180,E1 12077.155,E2 12077.155} C_VEL
LIN {X 0,Y 275.164,Z 357.679,A -85,B 0,C 180,E1 12073.876,E2 12073.876} C_VEL
LIN {X 0,Y 272.927,Z 353.563,A -85,B 0,C 180,E1 12070.554,E2 12070.554} C_VEL
LIN {X 0,Y 269.521,Z 347.651,A -85,B 0,C 180,E1 12063.402,E2 12063.402} C_VEL
LIN {X 0,Y 267.908,Z 346.09,A -85,B 0,C 180,E1 12057.433,E2 12057.433} C_VEL
LIN {X 0,Y 268.03,Z 346.237,A -85,B 0,C 180,E1 12052.066,E2 12052.066} C_VEL
LIN {X 0,Y 269.456,Z 347.833,A -85,B 0,C 180,E1 12046.917,E2 12046.917} C_VEL
LIN {X 0,Y 272.292,Z 353.128,A -85,B 0,C 180,E1 12040.478,E2 12040.478} C_VEL
LIN {X 0,Y 274.458,Z 357.249,A -85,B 0,C 180,E1 12036.944,E2 12036.944} C_VEL
LIN {X 0,Y 278.958,Z 362.732,A -85,B 0,C 180,E1 12034.069,E2 12034.069} C_VEL
LIN {X 0,Y 285.034,Z 370.137,A -85,B 0,C 180,E1 12030.869,E2 12030.869} C_VEL
LIN {X 0,Y 291.75,Z 378.69,A -85,B 0,C 180,E1 12027.83,E2 12027.83} C_VEL
LIN {X 0,Y 299.601,Z 389.586,A -85,B 0,C 180,E1 12024.735,E2 12024.735} C_VEL
LIN {X 0,Y 307.927,Z 401.985,A -85,B 0,C 180,E1 12021.847,E2 12021.847} C_VEL
LIN {X 0,Y 317.049,Z 417.21,A -85,B 0,C 180,E1 12019.007,E2 12019.007} C_VEL
LIN {X 0,Y 320.808,Z 424.476,A -85,B 0,C 180,E1 12017.903,E2 12017.903} C_VEL
LIN {X 0,Y 313.005,Z 571.897,A -85,B 0,C 180,E1 12014.768,E2 12014.768} C_VEL
LIN {X 0,Y 311.458,Z 591.638,A -85,B 0,C 180,E1 12014.067,E2 12014.067} C_VEL
LIN {X 0,Y 309.037,Z 610.166,A -85,B 0,C 180,E1 12013.114,E2 12013.114} C_VEL
LIN {X 0,Y 305.73,Z 628.487,A -85,B 0,C 180,E1 12011.847,E2 12011.847} C_VEL
LIN {X 0,Y 301.649,Z 646.164,A -85,B 0,C 180,E1 12010.266,E2 12010.266} C_VEL
LIN {X 0,Y 297.002,Z 662.734,A -85,B 0,C 180,E1 12008.397,E2 12008.397} C_VEL
LIN {X 0,Y 291.753,Z 678.821,A -85,B 0,C 180,E1 12006.117,E2 12006.117} C_VEL
LIN {X 0,Y 286.633,Z 692.662,A -85,B 0,C 180,E1 12003.685,E2 12003.685} C_VEL
LIN {X 0,Y 281.243,Z 705.935,A -85,B 0,C 180,E1 12000.792,E2 12000.792} C_VEL
LIN {X 0,Y 276.104,Z 717.629,A -85,B 0,C 180,E1 11997.614,E2 11997.614} C_VEL
LIN {X 0,Y 271.411,Z 727.804,A -85,B 0,C 180,E1 11994.136,E2 11994.136} C_VEL
LIN {X 0,Y 267.314,Z 736.464,A -85,B 0,C 180,E1 11990.356,E2 11990.356} C_VEL
LIN {X 0,Y 263.941,Z 743.582,A -85,B 0,C 180,E1 11986.279,E2 11986.279} C_VEL
LIN {X 0,Y 261.438,Z 749.087,A -85,B 0,C 180,E1 11981.918,E2 11981.918} C_VEL
LIN {X 0,Y 259.852,Z 752.75,A -85,B 0,C 180,E1 11977.517,E2 11977.517} C_VEL
LIN {X 0,Y 259.071,Z 754.711,A -85,B 0,C 180,E1 11973.097,E2 11973.097} C_VEL
LIN {X 0,Y 258.946,Z 755.052,A -85,B 0,C 180,E1 11968.673,E2 11968.673} C_VEL
LIN {X 0,Y 259.439,Z 753.792,A -85,B 0,C 180,E1 11964.249,E2 11964.249} C_VEL
LIN {X 0,Y 260.673,Z 750.871,A -85,B 0,C 180,E1 11959.838,E2 11959.838} C_VEL
LIN {X 0,Y 262.772,Z 746.174,A -85,B 0,C 180,E1 11955.456,E2 11955.456} C_VEL
LIN {X 0,Y 265.709,Z 739.912,A -85,B 0,C 180,E1 11951.347,E2 11951.347} C_VEL
LIN {X 0,Y 269.412,Z 732.169,A -85,B 0,C 180,E1 11947.527,E2 11947.527} C_VEL
LIN {X 0,Y 273.762,Z 722.884,A -85,B 0,C 180,E1 11943.958,E2 11943.958} C_VEL
LIN {X 0,Y 278.809,Z 711.732,A -85,B 0,C 180,E1 11940.575,E2 11940.575} C_VEL
LIN {X 0,Y 283.938,Z 699.648,A -85,B 0,C 180,E1 11937.64,E2 11937.64} C_VEL
LIN {X 0,Y 289.415,Z 685.558,A -85,B 0,C 180,E1 11934.886,E2 11934.886} C_VEL
LIN {X 0,Y 294.534,Z 670.895,A -85,B 0,C 180,E1 11932.581,E2 11932.581} C_VEL
LIN {X 0,Y 299.506,Z 654.524,A -85,B 0,C 180,E1 11930.51,E2 11930.51} C_VEL
LIN {X 0,Y 303.786,Z 637.887,A -85,B 0,C 180,E1 11928.834,E2 11928.834} C_VEL
LIN {X 0,Y 307.442,Z 620.315,A -85,B 0,C 180,E1 11927.434,E2 11927.434} C_VEL
LIN {X 0,Y 310.382,Z 601.677,A -85,B 0,C 180,E1 11926.301,E2 11926.301} C_VEL
LIN {X 0,Y 312.419,Z 582.429,A -85,B 0,C 180,E1 11925.456,E2 11925.456} C_VEL
LIN {X 0,Y 313.657,Z 560.196,A -85,B 0,C 180,E1 11924.83,E2 11924.83} C_VEL
LIN {X 0,Y 318.781,Z 462.892,A -85,B 0,C 180,E1 11922.784,E2 11922.784} C_VEL
LIN {X 0,Y 318.575,Z 455.305,A -85,B 0,C 180,E1 11922.489,E2 11922.489} C_VEL
LIN {X 0,Y 315.809,Z 435.494,A -85,B 0,C 180,E1 11921.194,E2 11921.194} C_VEL
LIN {X 0,Y 315.722,Z 428.973,A -85,B 0,C 180,E1 11920.948,E2 11920.948} C_VEL
LIN {X 0,Y 315.662,Z 427.477,A -85,B 0,C 180,E1 11920.881,E2 11920.881} C_VEL
LIN {X 0,Y 307.347,Z 412.836,A -85,B 0,C 180,E1 11918.268,E2 11918.268} C_VEL
LIN {X 0,Y 300.149,Z 401.392,A -85,B 0,C 180,E1 11915.777,E2 11915.777} C_VEL
LIN {X 0,Y 292.072,Z 389.55,A -85,B 0,C 180,E1 11912.636,E2 11912.636} C_VEL
LIN {X 0,Y 284.605,Z 379.682,A -85,B 0,C 180,E1 11909.289,E2 11909.289} C_VEL
LIN {X 0,Y 280.969,Z 375.046,A -85,B 0,C 180,E1 11907.442,E2 11907.442} C_VEL
LIN {X 0,Y 277.006,Z 370.123,A -85,B 0,C 180,E1 11905.21,E2 11905.21} C_VEL
LIN {X 0,Y 273.074,Z 365.247,A -85,B 0,C 180,E1 11902.68,E2 11902.68} C_VEL
LIN {X 0,Y 268.53,Z 360.386,A -85,B 0,C 180,E1 11899.241,E2 11899.241} C_VEL
LIN {X 0,Y 267.517,Z 359.038,A -85,B 0,C 180,E1 11898.298,E2 11898.298} C_VEL
LIN {X 0,Y 265.017,Z 354.234,A -85,B 0,C 180,E1 11891.756,E2 11891.756} C_VEL
LIN {X 0,Y 263.83,Z 353.036,A -85,B 0,C 180,E1 11885.655,E2 11885.655} C_VEL
LIN {X 0,Y 264.326,Z 353.564,A -85,B 0,C 180,E1 11880.217,E2 11880.217} C_VEL
LIN {X 0,Y 265.573,Z 354.883,A -85,B 0,C 180,E1 11876.331,E2 11876.331} C_VEL
LIN {X 0,Y 268.502,Z 360.09,A -85,B 0,C 180,E1 11869.921,E2 11869.921} C_VEL
LIN {X 0,Y 270.94,Z 364.479,A -85,B 0,C 180,E1 11866.339,E2 11866.339} C_VEL
LIN {X 0,Y 273.615,Z 369.146,A -85,B 0,C 180,E1 11863.44,E2 11863.44} C_VEL
LIN {X 0,Y 279.467,Z 376.816,A -85,B 0,C 180,E1 11859.858,E2 11859.858} C_VEL
LIN {X 0,Y 286.173,Z 386.133,A -85,B 0,C 180,E1 11856.419,E2 11856.419} C_VEL
LIN {X 0,Y 292.702,Z 395.716,A -85,B 0,C 180,E1 11853.527,E2 11853.527} C_VEL
LIN {X 0,Y 300.012,Z 407.122,A -85,B 0,C 180,E1 11850.666,E2 11850.666} C_VEL
LIN {X 0,Y 307.696,Z 420.322,A -85,B 0,C 180,E1 11847.963,E2 11847.963} C_VEL
LIN {X 0,Y 315.333,Z 434.737,A -85,B 0,C 180,E1 11845.502,E2 11845.502} C_VEL
LIN {X 0,Y 316.291,Z 437.142,A -85,B 0,C 180,E1 11845.188,E2 11845.188} C_VEL
LIN {X 0,Y 316.222,Z 443.384,A -85,B 0,C 180,E1 11844.968,E2 11844.968} C_VEL
LIN {X 0,Y 304.593,Z 622.097,A -85,B 0,C 180,E1 11840.822,E2 11840.822} C_VEL
LIN {X 0,Y 301.813,Z 643.788,A -85,B 0,C 180,E1 11840.049,E2 11840.049} C_VEL
LIN {X 0,Y 297.77,Z 665.007,A -85,B 0,C 180,E1 11838.995,E2 11838.995} C_VEL
LIN {X 0,Y 293.03,Z 684.694,A -85,B 0,C 180,E1 11837.673,E2 11837.673} C_VEL
LIN {X 0,Y 287.673,Z 703.642,A -85,B 0,C 180,E1 11836.009,E2 11836.009} C_VEL
LIN {X 0,Y 282.04,Z 721.457,A -85,B 0,C 180,E1 11834.013,E2 11834.013} C_VEL
LIN {X 0,Y 276.168,Z 738.482,A -85,B 0,C 180,E1 11831.631,E2 11831.631} C_VEL
LIN {X 0,Y 270.255,Z 754.629,A -85,B 0,C 180,E1 11828.835,E2 11828.835} C_VEL
LIN {X 0,Y 264.61,Z 769.797,A -85,B 0,C 180,E1 11825.583,E2 11825.583} C_VEL
LIN {X 0,Y 259.425,Z 783.837,A -85,B 0,C 180,E1 11821.87,E2 11821.87} C_VEL
LIN {X 0,Y 255.163,Z 796.286,A -85,B 0,C 180,E1 11817.794,E2 11817.794} C_VEL
LIN {X 0,Y 251.974,Z 807.122,A -85,B 0,C 180,E1 11813.378,E2 11813.378} C_VEL
LIN {X 0,Y 250.049,Z 815.871,A -85,B 0,C 180,E1 11808.898,E2 11808.898} C_VEL
LIN {X 0,Y 249.253,Z 822.73,A -85,B 0,C 180,E1 11804.401,E2 11804.401} C_VEL
LIN {X 0,Y 249.312,Z 827.793,A -85,B 0,C 180,E1 11799.93,E2 11799.93} C_VEL
LIN {X 0,Y 249.832,Z 830.863,A -85,B 0,C 180,E1 11795.742,E2 11795.742} C_VEL
LIN {X 0,Y 250.258,Z 832.286,A -85,B 0,C 180,E1 11792.061,E2 11792.061} C_VEL
LIN {X 0,Y 250.319,Z 832.404,A -85,B 0,C 180,E1 11788.856,E2 11788.856} C_VEL
LIN {X 0,Y 249.956,Z 831.366,A -85,B 0,C 180,E1 11785.181,E2 11785.181} C_VEL
LIN {X 0,Y 249.439,Z 828.746,A -85,B 0,C 180,E1 11781.239,E2 11781.239} C_VEL
LIN {X 0,Y 249.193,Z 824.191,A -85,B 0,C 180,E1 11776.779,E2 11776.779} C_VEL
LIN {X 0,Y 249.74,Z 817.851,A -85,B 0,C 180,E1 11772.286,E2 11772.286} C_VEL
LIN {X 0,Y 251.355,Z 809.631,A -85,B 0,C 180,E1 11767.797,E2 11767.797} C_VEL
LIN {X 0,Y 254.195,Z 799.352,A -85,B 0,C 180,E1 11763.359,E2 11763.359} C_VEL
LIN {X 0,Y 258.116,Z 787.497,A -85,B 0,C 180,E1 11759.249,E2 11759.249} C_VEL
LIN {X 0,Y 262.962,Z 774.122,A -85,B 0,C 180,E1 11755.492,E2 11755.492} C_VEL
LIN {X 0,Y 268.385,Z 759.548,A -85,B 0,C 180,E1 11752.166,E2 11752.166} C_VEL
LIN {X 0,Y 274.179,Z 743.815,A -85,B 0,C 180,E1 11749.251,E2 11749.251} C_VEL
LIN {X 0,Y 280.09,Z 727.014,A -85,B 0,C 180,E1 11746.735,E2 11746.735} C_VEL
LIN {X 0,Y 285.816,Z 709.369,A -85,B 0,C 180,E1 11744.612,E2 11744.612} C_VEL
LIN {X 0,Y 291.483,Z 689.924,A -85,B 0,C 180,E1 11742.773,E2 11742.773} C_VEL
LIN {X 0,Y 296.536,Z 669.888,A -85,B 0,C 180,E1 11741.326,E2 11741.326} C_VEL
LIN {X 0,Y 300.808,Z 648.932,A -85,B 0,C 180,E1 11740.204,E2 11740.204} C_VEL
LIN {X 0,Y 303.908,Z 627.285,A -85,B 0,C 180,E1 11739.364,E2 11739.364} C_VEL
LIN {X 0,Y 306.061,Z 599.729,A -85,B 0,C 180,E1 11738.64,E2 11738.64} C_VEL
LIN {X 0,Y 316.255,Z 439.472,A -85,B 0,C 180,E1 11734.937,E2 11734.937} C_VEL
LIN {X 0,Y 315.971,Z 436.213,A -85,B 0,C 180,E1 11734.749,E2 11734.749} C_VEL
LIN {X 0,Y 308.414,Z 421.704,A -85,B 0,C 180,E1 11732.338,E2 11732.338} C_VEL
LIN {X 0,Y 300.211,Z 407.543,A -85,B 0,C 180,E1 11729.477,E2 11729.477} C_VEL
LIN {X 0,Y 292.84,Z 396.03,A -85,B 0,C 180,E1 11726.624,E2 11726.624} C_VEL
LIN {X 0,Y 287.054,Z 387.519,A -85,B 0,C 180,E1 11724.104,E2 11724.104} C_VEL
LIN {X 0,Y 283.294,Z 382.254,A -85,B 0,C 180,E1 11722.297,E2 11722.297} C_VEL
LIN {X 0,Y 277.653,Z 374.456,A -85,B 0,C 180,E1 11719.238,E2 11719.238} C_VEL
LIN {X 0,Y 273.404,Z 368.944,A -85,B 0,C 180,E1 11716.573,E2 11716.573} C_VEL
LIN {X 0,Y 270.804,Z 364.328,A -85,B 0,C 180,E1 11713.668,E2 11713.668} C_VEL
LIN {X 0,Y 268.482,Z 360.116,A -85,B 0,C 180,E1 11710.297,E2 11710.297} C_VEL
LIN {X 0,Y 265.269,Z 354.401,A -85,B 0,C 180,E1 11703.241,E2 11703.241} C_VEL
LIN {X 0,Y 263.711,Z 352.868,A -85,B 0,C 180,E1 11696.957,E2 11696.957} C_VEL
LIN {X 0,Y 263.979,Z 353.221,A -85,B 0,C 180,E1 11691.285,E2 11691.285} C_VEL
LIN {X 0,Y 265.225,Z 354.68,A -85,B 0,C 180,E1 11686.927,E2 11686.927} C_VEL
LIN {X 0,Y 267.657,Z 359.152,A -85,B 0,C 180,E1 11681.26,E2 11681.26} C_VEL
LIN {X 0,Y 272.055,Z 364.369,A -85,B 0,C 180,E1 11677.756,E2 11677.756} C_VEL
LIN {X 0,Y 273.384,Z 365.807,A -85,B 0,C 180,E1 11676.848,E2 11676.848} C_VEL
LIN {X 0,Y 277.358,Z 370.442,A -85,B 0,C 180,E1 11674.367,E2 11674.367} C_VEL
LIN {X 0,Y 282.945,Z 377.568,A -85,B 0,C 180,E1 11671.333,E2 11671.333} C_VEL
LIN {X 0,Y 289.194,Z 385.686,A -85,B 0,C 180,E1 11668.412,E2 11668.412} C_VEL
LIN {X 0,Y 296.958,Z 396.688,A -85,B 0,C 180,E1 11665.251,E2 11665.251} C_VEL
LIN {X 0,Y 305.116,Z 409.234,A -85,B 0,C 180,E1 11662.326,E2 11662.326} C_VEL
LIN {X 0,Y 313.511,Z 423.635,A -85,B 0,C 180,E1 11659.623,E2 11659.623} C_VEL
LIN {X 0,Y 315.646,Z 427.98,A -85,B 0,C 180,E1 11658.962,E2 11658.962} C_VEL
LIN {X 0,Y 307.654,Z 572.466,A -85,B 0,C 180,E1 11655.861,E2 11655.861} C_VEL
LIN {X 0,Y 306.034,Z 592.378,A -85,B 0,C 180,E1 11655.15,E2 11655.15} C_VEL
LIN {X 0,Y 303.473,Z 611.223,A -85,B 0,C 180,E1 11654.172,E2 11654.172} C_VEL
LIN {X 0,Y 299.921,Z 630.065,A -85,B 0,C 180,E1 11652.849,E2 11652.849} C_VEL
LIN {X 0,Y 295.686,Z 647.616,A -85,B 0,C 180,E1 11651.252,E2 11651.252} C_VEL
LIN {X 0,Y 290.843,Z 664.176,A -85,B 0,C 180,E1 11649.352,E2 11649.352} C_VEL
LIN {X 0,Y 285.626,Z 679.555,A -85,B 0,C 180,E1 11647.145,E2 11647.145} C_VEL
LIN {X 0,Y 280.092,Z 693.944,A -85,B 0,C 180,E1 11644.581,E2 11644.581} C_VEL
LIN {X 0,Y 274.476,Z 707.191,A -85,B 0,C 180,E1 11641.638,E2 11641.638} C_VEL
LIN {X 0,Y 269.11,Z 718.867,A -85,B 0,C 180,E1 11638.396,E2 11638.396} C_VEL
LIN {X 0,Y 264.194,Z 729.029,A -85,B 0,C 180,E1 11634.839,E2 11634.839} C_VEL
LIN {X 0,Y 259.891,Z 737.68,A -85,B 0,C 180,E1 11630.964,E2 11630.964} C_VEL
LIN {X 0,Y 256.336,Z 744.792,A -85,B 0,C 180,E1 11626.776,E2 11626.776} C_VEL
LIN {X 0,Y 253.686,Z 750.293,A -85,B 0,C 180,E1 11622.288,E2 11622.288} C_VEL
LIN {X 0,Y 252.003,Z 753.954,A -85,B 0,C 180,E1 11617.753,E2 11617.753} C_VEL
LIN {X 0,Y 251.171,Z 755.913,A -85,B 0,C 180,E1 11613.195,E2 11613.195} C_VEL
LIN {X 0,Y 251.039,Z 756.254,A -85,B 0,C 180,E1 11608.631,E2 11608.631} C_VEL
LIN {X 0,Y 251.564,Z 754.995,A -85,B 0,C 180,E1 11604.069,E2 11604.069} C_VEL
LIN {X 0,Y 252.876,Z 752.076,A -85,B 0,C 180,E1 11599.521,E2 11599.521} C_VEL
LIN {X 0,Y 255.102,Z 747.382,A -85,B 0,C 180,E1 11595.009,E2 11595.009} C_VEL
LIN {X 0,Y 258.204,Z 741.123,A -85,B 0,C 180,E1 11590.783,E2 11590.783} C_VEL
LIN {X 0,Y 262.173,Z 733.239,A -85,B 0,C 180,E1 11586.798,E2 11586.798} C_VEL
LIN {X 0,Y 266.893,Z 723.638,A -85,B 0,C 180,E1 11583.045,E2 11583.045} C_VEL
LIN {X 0,Y 271.94,Z 712.971,A -85,B 0,C 180,E1 11579.755,E2 11579.755} C_VEL
LIN {X 0,Y 277.289,Z 700.908,A -85,B 0,C 180,E1 11576.765,E2 11576.765} C_VEL
LIN {X 0,Y 282.99,Z 686.848,A -85,B 0,C 180,E1 11573.966,E2 11573.966} C_VEL
LIN {X 0,Y 288.434,Z 671.864,A -85,B 0,C 180,E1 11571.577,E2 11571.577} C_VEL
LIN {X 0,Y 293.469,Z 655.921,A -85,B 0,C 180,E1 11569.532,E2 11569.532} C_VEL
LIN {X 0,Y 298.059,Z 638.753,A -85,B 0,C 180,E1 11567.781,E2 11567.781} C_VEL
LIN {X 0,Y 301.939,Z 620.702,A -85,B 0,C 180,E1 11566.337,E2 11566.337} C_VEL
LIN {X 0,Y 305.048,Z 601.447,A -85,B 0,C 180,E1 11565.171,E2 11565.171} C_VEL
LIN {X 0,Y 307.146,Z 581.799,A -85,B 0,C 180,E1 11564.321,E2 11564.321} C_VEL
LIN {X 0,Y 308.502,Z 557.357,A -85,B 0,C 180,E1 11563.657,E2 11563.657} C_VEL
LIN {X 0,Y 315.722,Z 428.973,A -85,B 0,C 180,E1 11560.948,E2 11560.948} C_VEL
LIN {X 0,Y 315.453,Z 426.101,A -85,B 0,C 180,E1 11560.784,E2 11560.784} C_VEL
LIN {X 0,Y 314.164,Z 422.942,A -85,B 0,C 180,E1 11560.365,E2 11560.365} C_VEL
LIN {X 0,Y 311.128,Z 419.574,A -85,B 0,C 180,E1 11559.498,E2 11559.498} C_VEL
LIN {X 0,Y 301.539,Z 414.029,A -85,B 0,C 180,E1 11556.707,E2 11556.707} C_VEL
LIN {X 0,Y 299.386,Z 411.597,A -85,B 0,C 180,E1 11555.977,E2 11555.977} C_VEL
LIN {X 0,Y 291.54,Z 399.548,A -85,B 0,C 180,E1 11552.929,E2 11552.929} C_VEL
LIN {X 0,Y 283.395,Z 388.069,A -85,B 0,C 180,E1 11549.252,E2 11549.252} C_VEL
LIN {X 0,Y 278.605,Z 382.043,A -85,B 0,C 180,E1 11546.77,E2 11546.77} C_VEL
LIN {X 0,Y 274.918,Z 377.366,A -85,B 0,C 180,E1 11544.604,E2 11544.604} C_VEL
LIN {X 0,Y 270.738,Z 372.222,A -85,B 0,C 180,E1 11541.787,E2 11541.787} C_VEL
LIN {X 0,Y 266.769,Z 367.583,A -85,B 0,C 180,E1 11538.578,E2 11538.578} C_VEL
LIN {X 0,Y 260.852,Z 361.011,A -85,B 0,C 180,E1 11531.498,E2 11531.498} C_VEL
LIN {X 0,Y 259.657,Z 359.856,A -85,B 0,C 180,E1 11525.525,E2 11525.525} C_VEL
LIN {X 0,Y 260.201,Z 360.429,A -85,B 0,C 180,E1 11520,E2 11520} C_VEL
LIN {X 0,Y 261.322,Z 361.624,A -85,B 0,C 180,E1 11516.491,E2 11516.491} C_VEL
LIN {X 0,Y 264.546,Z 367.06,A -85,B 0,C 180,E1 11510.098,E2 11510.098} C_VEL
LIN {X 0,Y 268.091,Z 371.757,A -85,B 0,C 180,E1 11506.751,E2 11506.751} C_VEL
LIN {X 0,Y 273.021,Z 378.307,A -85,B 0,C 180,E1 11503.074,E2 11503.074} C_VEL
LIN {X 0,Y 277.486,Z 384.308,A -85,B 0,C 180,E1 11500.312,E2 11500.312} C_VEL
LIN {X 0,Y 283.769,Z 393.268,A -85,B 0,C 180,E1 11496.977,E2 11496.977} C_VEL
LIN {X 0,Y 289.947,Z 402.565,A -85,B 0,C 180,E1 11494.137,E2 11494.137} C_VEL
LIN {X 0,Y 297.098,Z 414.031,A -85,B 0,C 180,E1 11491.233,E2 11491.233} C_VEL
LIN {X 0,Y 305.535,Z 428.951,A -85,B 0,C 180,E1 11488.179,E2 11488.179} C_VEL
LIN {X 0,Y 311.41,Z 440.745,A -85,B 0,C 180,E1 11486.205,E2 11486.205} C_VEL
LIN {X 0,Y 299.939,Z 613.756,A -85,B 0,C 180,E1 11482.177,E2 11482.177} C_VEL
LIN {X 0,Y 297.737,Z 634.349,A -85,B 0,C 180,E1 11481.537,E2 11481.537} C_VEL
LIN {X 0,Y 294.375,Z 654.325,A -85,B 0,C 180,E1 11480.673,E2 11480.673} C_VEL
LIN {X 0,Y 289.873,Z 674.284,A -85,B 0,C 180,E1 11479.512,E2 11479.512} C_VEL
LIN {X 0,Y 284.573,Z 693.791,A -85,B 0,C 180,E1 11477.995,E2 11477.995} C_VEL
LIN {X 0,Y 278.62,Z 712.855,A -85,B 0,C 180,E1 11476.067,E2 11476.067} C_VEL
LIN {X 0,Y 272.428,Z 730.666,A -85,B 0,C 180,E1 11473.773,E2 11473.773} C_VEL
LIN {X 0,Y 266.189,Z 747.277,A -85,B 0,C 180,E1 11471.095,E2 11471.095} C_VEL
LIN {X 0,Y 260.188,Z 762.629,A -85,B 0,C 180,E1 11468.022,E2 11468.022} C_VEL
LIN {X 0,Y 254.823,Z 776.222,A -85,B 0,C 180,E1 11464.675,E2 11464.675} C_VEL
LIN {X 0,Y 249.934,Z 789.048,A -85,B 0,C 180,E1 11460.8,E2 11460.8} C_VEL
LIN {X 0,Y 245.999,Z 800.41,A -85,B 0,C 180,E1 11456.556,E2 11456.556} C_VEL
LIN {X 0,Y 243.195,Z 810.243,A -85,B 0,C 180,E1 11451.97,E2 11451.97} C_VEL
LIN {X 0,Y 241.661,Z 818.097,A -85,B 0,C 180,E1 11447.331,E2 11447.331} C_VEL
LIN {X 0,Y 241.215,Z 824.117,A -85,B 0,C 180,E1 11442.69,E2 11442.69} C_VEL
LIN {X 0,Y 241.538,Z 828.112,A -85,B 0,C 180,E1 11438.33,E2 11438.33} C_VEL
LIN {X 0,Y 242.114,Z 830.426,A -85,B 0,C 180,E1 11434.263,E2 11434.263} C_VEL
LIN {X 0,Y 242.425,Z 831.259,A -85,B 0,C 180,E1 11430.709,E2 11430.709} C_VEL
LIN {X 0,Y 242.269,Z 830.908,A -85,B 0,C 180,E1 11427.123,E2 11427.123} C_VEL
LIN {X 0,Y 241.766,Z 829.214,A -85,B 0,C 180,E1 11423.35,E2 11423.35} C_VEL
LIN {X 0,Y 241.279,Z 825.816,A -85,B 0,C 180,E1 11419.011,E2 11419.011} C_VEL
LIN {X 0,Y 241.392,Z 820.517,A -85,B 0,C 180,E1 11414.382,E2 11414.382} C_VEL
LIN {X 0,Y 242.576,Z 812.939,A -85,B 0,C 180,E1 11409.491,E2 11409.491} C_VEL
LIN {X 0,Y 244.961,Z 803.735,A -85,B 0,C 180,E1 11404.882,E2 11404.882} C_VEL
LIN {X 0,Y 248.487,Z 793.032,A -85,B 0,C 180,E1 11400.601,E2 11400.601} C_VEL
LIN {X 0,Y 252.959,Z 780.921,A -85,B 0,C 180,E1 11396.674,E2 11396.674} C_VEL
LIN {X 0,Y 258.222,Z 767.453,A -85,B 0,C 180,E1 11393.119,E2 11393.119} C_VEL
LIN {X 0,Y 264.176,Z 752.263,A -85,B 0,C 180,E1 11389.865,E2 11389.865} C_VEL
LIN {X 0,Y 270.488,Z 735.645,A -85,B 0,C 180,E1 11387.001,E2 11387.001} C_VEL
LIN {X 0,Y 276.674,Z 718.278,A -85,B 0,C 180,E1 11384.61,E2 11384.61} C_VEL
LIN {X 0,Y 282.584,Z 700.006,A -85,B 0,C 180,E1 11382.613,E2 11382.613} C_VEL
LIN {X 0,Y 287.937,Z 681.319,A -85,B 0,C 180,E1 11381.018,E2 11381.018} C_VEL
LIN {X 0,Y 292.634,Z 662.062,A -85,B 0,C 180,E1 11379.758,E2 11379.758} C_VEL
LIN {X 0,Y 296.561,Z 641.568,A -85,B 0,C 180,E1 11378.763,E2 11378.763} C_VEL
LIN {X 0,Y 299.288,Z 620.33,A -85,B 0,C 180,E1 11378.017,E2 11378.017} C_VEL
LIN {X 0,Y 311.297,Z 441.152,A -85,B 0,C 180,E1 11373.832,E2 11373.832} C_VEL
LIN {X 0,Y 310.816,Z 439.448,A -85,B 0,C 180,E1 11373.649,E2 11373.649} C_VEL
LIN {X 0,Y 302.479,Z 423.487,A -85,B 0,C 180,E1 11370.821,E2 11370.821} C_VEL
LIN {X 0,Y 294.957,Z 410.543,A -85,B 0,C 180,E1 11368.001,E2 11368.001} C_VEL
LIN {X 0,Y 287.632,Z 398.981,A -85,B 0,C 180,E1 11364.928,E2 11364.928} C_VEL
LIN {X 0,Y 281.321,Z 389.864,A -85,B 0,C 180,E1 11361.912,E2 11361.912} C_VEL
LIN {X 0,Y 275.621,Z 381.795,A -85,B 0,C 180,E1 11358.726,E2 11358.726} C_VEL
LIN {X 0,Y 271.339,Z 376.126,A -85,B 0,C 180,E1 11355.933,E2 11355.933} C_VEL
LIN {X 0,Y 267.869,Z 371.581,A -85,B 0,C 180,E1 11353.271,E2 11353.271} C_VEL
LIN {X 0,Y 264.423,Z 366.898,A -85,B 0,C 180,E1 11350.016,E2 11350.016} C_VEL
LIN {X 0,Y 261.036,Z 361.164,A -85,B 0,C 180,E1 11343.073,E2 11343.073} C_VEL
LIN {X 0,Y 259.523,Z 359.666,A -85,B 0,C 180,E1 11336.687,E2 11336.687} C_VEL
LIN {X 0,Y 259.871,Z 360.112,A -85,B 0,C 180,E1 11330.923,E2 11330.923} C_VEL
LIN {X 0,Y 261.203,Z 361.397,A -85,B 0,C 180,E1 11327.397,E2 11327.397} C_VEL
LIN {X 0,Y 265.33,Z 366.168,A -85,B 0,C 180,E1 11322.433,E2 11322.433} C_VEL
LIN {X 0,Y 266.687,Z 367.503,A -85,B 0,C 180,E1 11321.19,E2 11321.19} C_VEL
LIN {X 0,Y 270.552,Z 372.073,A -85,B 0,C 180,E1 11318.083,E2 11318.083} C_VEL
LIN {X 0,Y 271.984,Z 373.859,A -85,B 0,C 180,E1 11317.065,E2 11317.065} C_VEL
LIN {X 0,Y 276.235,Z 379.016,A -85,B 0,C 180,E1 11314.371,E2 11314.371} C_VEL
LIN {X 0,Y 280.703,Z 384.74,A -85,B 0,C 180,E1 11311.896,E2 11311.896} C_VEL
LIN {X 0,Y 286.718,Z 392.744,A -85,B 0,C 180,E1 11308.986,E2 11308.986} C_VEL
LIN {X 0,Y 294.761,Z 404.38,A -85,B 0,C 180,E1 11305.612,E2 11305.612} C_VEL
LIN {X 0,Y 303.115,Z 417.764,A -85,B 0,C 180,E1 11302.541,E2 11302.541} C_VEL
LIN {X 0,Y 310.604,Z 431.188,A -85,B 0,C 180,E1 11300.064,E2 11300.064} C_VEL
LIN {X 0,Y 302.407,Z 573.246,A -85,B 0,C 180,E1 11296.987,E2 11296.987} C_VEL
LIN {X 0,Y 300.706,Z 593.258,A -85,B 0,C 180,E1 11296.265,E2 11296.265} C_VEL
LIN {X 0,Y 298.016,Z 612.277,A -85,B 0,C 180,E1 11295.268,E2 11295.268} C_VEL
LIN {X 0,Y 294.452,Z 630.537,A -85,B 0,C 180,E1 11293.979,E2 11293.979} C_VEL
LIN {X 0,Y 290.057,Z 648.192,A -85,B 0,C 180,E1 11292.368,E2 11292.368} C_VEL
LIN {X 0,Y 284.883,Z 665.271,A -85,B 0,C 180,E1 11290.393,E2 11290.393} C_VEL
LIN {X 0,Y 279.376,Z 680.87,A -85,B 0,C 180,E1 11288.122,E2 11288.122} C_VEL
LIN {X 0,Y 273.622,Z 695.221,A -85,B 0,C 180,E1 11285.521,E2 11285.521} C_VEL
LIN {X 0,Y 267.772,Z 708.444,A -85,B 0,C 180,E1 11282.526,E2 11282.526} C_VEL
LIN {X 0,Y 262.169,Z 720.104,A -85,B 0,C 180,E1 11279.219,E2 11279.219} C_VEL
LIN {X 0,Y 257.021,Z 730.255,A -85,B 0,C 180,E1 11275.582,E2 11275.582} C_VEL
LIN {X 0,Y 252.501,Z 738.898,A -85,B 0,C 180,E1 11271.608,E2 11271.608} C_VEL
LIN {X 0,Y 248.751,Z 746.004,A -85,B 0,C 180,E1 11267.304,E2 11267.304} C_VEL
LIN {X 0,Y 245.944,Z 751.501,A -85,B 0,C 180,E1 11262.681,E2 11262.681} C_VEL
LIN {X 0,Y 244.158,Z 755.158,A -85,B 0,C 180,E1 11258.003,E2 11258.003} C_VEL
LIN {X 0,Y 243.272,Z 757.115,A -85,B 0,C 180,E1 11253.299,E2 11253.299} C_VEL
LIN {X 0,Y 243.132,Z 757.455,A -85,B 0,C 180,E1 11248.586,E2 11248.586} C_VEL
LIN {X 0,Y 243.691,Z 756.197,A -85,B 0,C 180,E1 11243.876,E2 11243.876} C_VEL
LIN {X 0,Y 245.087,Z 753.28,A -85,B 0,C 180,E1 11239.184,E2 11239.184} C_VEL
LIN {X 0,Y 247.447,Z 748.588,A -85,B 0,C 180,E1 11234.533,E2 11234.533} C_VEL
LIN {X 0,Y 250.725,Z 742.333,A -85,B 0,C 180,E1 11230.187,E2 11230.187} C_VEL
LIN {X 0,Y 255.002,Z 734.264,A -85,B 0,C 180,E1 11226.008,E2 11226.008} C_VEL
LIN {X 0,Y 259.856,Z 724.856,A -85,B 0,C 180,E1 11222.25,E2 11222.25} C_VEL
LIN {X 0,Y 265.196,Z 714.075,A -85,B 0,C 180,E1 11218.855,E2 11218.855} C_VEL
LIN {X 0,Y 270.812,Z 701.935,A -85,B 0,C 180,E1 11215.795,E2 11215.795} C_VEL
LIN {X 0,Y 276.596,Z 688.252,A -85,B 0,C 180,E1 11213.025,E2 11213.025} C_VEL
LIN {X 0,Y 282.168,Z 673.561,A -85,B 0,C 180,E1 11210.634,E2 11210.634} C_VEL
LIN {X 0,Y 287.521,Z 657.318,A -85,B 0,C 180,E1 11208.513,E2 11208.513} C_VEL
LIN {X 0,Y 292.369,Z 639.895,A -85,B 0,C 180,E1 11206.712,E2 11206.712} C_VEL
LIN {X 0,Y 296.306,Z 622.353,A -85,B 0,C 180,E1 11205.288,E2 11205.288} C_VEL
LIN {X 0,Y 299.493,Z 603.691,A -85,B 0,C 180,E1 11204.131,E2 11204.131} C_VEL
LIN {X 0,Y 301.707,Z 584.601,A -85,B 0,C 180,E1 11203.27,E2 11203.27} C_VEL
LIN {X 0,Y 303.053,Z 563.144,A -85,B 0,C 180,E1 11202.641,E2 11202.641} C_VEL
LIN {X 0,Y 310.65,Z 431.116,A -85,B 0,C 180,E1 11199.8,E2 11199.8} C_VEL
LIN {X 0,Y 302.651,Z 416.894,A -85,B 0,C 180,E1 11197.139,E2 11197.139} C_VEL
LIN {X 0,Y 299.386,Z 411.597,A -85,B 0,C 180,E1 11195.977,E2 11195.977} C_VEL
LIN {X 0,Y 296.103,Z 407.989,A -85,B 0,C 180,E1 11194.815,E2 11194.815} C_VEL
LIN {X 0,Y 288.445,Z 403.386,A -85,B 0,C 180,E1 11192.017,E2 11192.017} C_VEL
LIN {X 0,Y 284.803,Z 400.362,A -85,B 0,C 180,E1 11190.49,E2 11190.49} C_VEL
LIN {X 0,Y 284.011,Z 399.335,A -85,B 0,C 180,E1 11190.122,E2 11190.122} C_VEL
LIN {X 0,Y 277.331,Z 390.187,A -85,B 0,C 180,E1 11186.671,E2 11186.671} C_VEL
LIN {X 0,Y 273.037,Z 384.773,A -85,B 0,C 180,E1 11184.099,E2 11184.099} C_VEL
LIN {X 0,Y 268.964,Z 379.69,A -85,B 0,C 180,E1 11181.251,E2 11181.251} C_VEL
LIN {X 0,Y 264.482,Z 374.303,A -85,B 0,C 180,E1 11177.377,E2 11177.377} C_VEL
LIN {X 0,Y 259.636,Z 368.814,A -85,B 0,C 180,E1 11171.102,E2 11171.102} C_VEL
LIN {X 0,Y 257.497,Z 367.549,A -85,B 0,C 180,E1 11164.901,E2 11164.901} C_VEL
LIN {X 0,Y 258.026,Z 368.268,A -85,B 0,C 180,E1 11159.112,E2 11159.112} C_VEL
LIN {X 0,Y 259.052,Z 369.438,A -85,B 0,C 180,E1 11156.46,E2 11156.46} C_VEL
LIN {X 0,Y 263.131,Z 374.76,A -85,B 0,C 180,E1 11150.486,E2 11150.486} C_VEL
LIN {X 0,Y 266.716,Z 379.556,A -85,B 0,C 180,E1 11147.002,E2 11147.002} C_VEL
LIN {X 0,Y 271.243,Z 385.883,A -85,B 0,C 180,E1 11143.511,E2 11143.511} C_VEL
LIN {X 0,Y 275.28,Z 391.416,A -85,B 0,C 180,E1 11140.92,E2 11140.92} C_VEL
LIN {X 0,Y 281.392,Z 400.399,A -85,B 0,C 180,E1 11137.544,E2 11137.544} C_VEL
LIN {X 0,Y 287.329,Z 409.57,A -85,B 0,C 180,E1 11134.714,E2 11134.714} C_VEL
LIN {X 0,Y 294.659,Z 421.67,A -85,B 0,C 180,E1 11131.637,E2 11131.637} C_VEL
LIN {X 0,Y 302.459,Z 436.06,A -85,B 0,C 180,E1 11128.707,E2 11128.707} C_VEL
LIN {X 0,Y 306.465,Z 444.425,A -85,B 0,C 180,E1 11127.295,E2 11127.295} C_VEL
LIN {X 0,Y 294.167,Z 620.486,A -85,B 0,C 180,E1 11123.171,E2 11123.171} C_VEL
LIN {X 0,Y 291.22,Z 642.131,A -85,B 0,C 180,E1 11122.394,E2 11122.394} C_VEL
LIN {X 0,Y 287.038,Z 662.887,A -85,B 0,C 180,E1 11121.363,E2 11121.363} C_VEL
LIN {X 0,Y 281.883,Z 682.993,A -85,B 0,C 180,E1 11120.009,E2 11120.009} C_VEL
LIN {X 0,Y 275.966,Z 702.468,A -85,B 0,C 180,E1 11118.274,E2 11118.274} C_VEL
LIN {X 0,Y 269.637,Z 720.875,A -85,B 0,C 180,E1 11116.155,E2 11116.155} C_VEL
LIN {X 0,Y 263.056,Z 738.26,A -85,B 0,C 180,E1 11113.618,E2 11113.618} C_VEL
LIN {X 0,Y 256.451,Z 754.612,A -85,B 0,C 180,E1 11110.624,E2 11110.624} C_VEL
LIN {X 0,Y 250.498,Z 768.957,A -85,B 0,C 180,E1 11107.35,E2 11107.35} C_VEL
LIN {X 0,Y 245.055,Z 782.1,A -85,B 0,C 180,E1 11103.66,E2 11103.66} C_VEL
LIN {X 0,Y 240.296,Z 794.336,A -85,B 0,C 180,E1 11099.405,E2 11099.405} C_VEL
LIN {X 0,Y 236.778,Z 804.563,A -85,B 0,C 180,E1 11094.978,E2 11094.978} C_VEL
LIN {X 0,Y 234.442,Z 813.342,A -85,B 0,C 180,E1 11090.209,E2 11090.209} C_VEL
LIN {X 0,Y 233.388,Z 820.231,A -85,B 0,C 180,E1 11085.403,E2 11085.403} C_VEL
LIN {X 0,Y 233.343,Z 825.326,A -85,B 0,C 180,E1 11080.617,E2 11080.617} C_VEL
LIN {X 0,Y 233.866,Z 828.29,A -85,B 0,C 180,E1 11076.382,E2 11076.382} C_VEL
LIN {X 0,Y 234.393,Z 829.845,A -85,B 0,C 180,E1 11072.445,E2 11072.445} C_VEL
LIN {X 0,Y 234.505,Z 830.027,A -85,B 0,C 180,E1 11069.023,E2 11069.023} C_VEL
LIN {X 0,Y 234.129,Z 829.119,A -85,B 0,C 180,E1 11065.346,E2 11065.346} C_VEL
LIN {X 0,Y 233.501,Z 826.48,A -85,B 0,C 180,E1 11060.884,E2 11060.884} C_VEL
LIN {X 0,Y 233.278,Z 821.992,A -85,B 0,C 180,E1 11056.112,E2 11056.112} C_VEL
LIN {X 0,Y 233.979,Z 815.722,A -85,B 0,C 180,E1 11051.308,E2 11051.308} C_VEL
LIN {X 0,Y 235.899,Z 807.55,A -85,B 0,C 180,E1 11046.521,E2 11046.521} C_VEL
LIN {X 0,Y 239.182,Z 797.347,A -85,B 0,C 180,E1 11041.812,E2 11041.812} C_VEL
LIN {X 0,Y 243.627,Z 785.587,A -85,B 0,C 180,E1 11037.478,E2 11037.478} C_VEL
LIN {X 0,Y 248.697,Z 773.145,A -85,B 0,C 180,E1 11033.773,E2 11033.773} C_VEL
LIN {X 0,Y 254.544,Z 759.011,A -85,B 0,C 180,E1 11030.344,E2 11030.344} C_VEL
LIN {X 0,Y 260.913,Z 743.411,A -85,B 0,C 180,E1 11027.291,E2 11027.291} C_VEL
LIN {X 0,Y 267.509,Z 726.344,A -85,B 0,C 180,E1 11024.617,E2 11024.617} C_VEL
LIN {X 0,Y 273.686,Z 708.928,A -85,B 0,C 180,E1 11022.443,E2 11022.443} C_VEL
LIN {X 0,Y 279.444,Z 690.889,A -85,B 0,C 180,E1 11020.666,E2 11020.666} C_VEL
LIN {X 0,Y 284.678,Z 672.092,A -85,B 0,C 180,E1 11019.231,E2 11019.231} C_VEL
LIN {X 0,Y 289.362,Z 651.581,A -85,B 0,C 180,E1 11018.059,E2 11018.059} C_VEL
LIN {X 0,Y 292.884,Z 630.334,A -85,B 0,C 180,E1 11017.17,E2 11017.17} C_VEL
LIN {X 0,Y 295.042,Z 608.532,A -85,B 0,C 180,E1 11016.533,E2 11016.533} C_VEL
LIN {X 0,Y 306.312,Z 443.938,A -85,B 0,C 180,E1 11012.698,E2 11012.698} C_VEL
LIN {X 0,Y 298.667,Z 429.025,A -85,B 0,C 180,E1 11009.976,E2 11009.976} C_VEL
LIN {X 0,Y 291.575,Z 416.554,A -85,B 0,C 180,E1 11007.189,E2 11007.189} C_VEL
LIN {X 0,Y 284.887,Z 405.688,A -85,B 0,C 180,E1 11004.244,E2 11004.244} C_VEL
LIN {X 0,Y 278.845,Z 396.729,A -85,B 0,C 180,E1 11001.232,E2 11001.232} C_VEL
LIN {X 0,Y 273.307,Z 388.764,A -85,B 0,C 180,E1 10998.006,E2 10998.006} C_VEL
LIN {X 0,Y 269.459,Z 383.477,A -85,B 0,C 180,E1 10995.385,E2 10995.385} C_VEL
LIN {X 0,Y 266.219,Z 379.13,A -85,B 0,C 180,E1 10992.802,E2 10992.802} C_VEL
LIN {X 0,Y 262.412,Z 373.892,A -85,B 0,C 180,E1 10988.987,E2 10988.987} C_VEL
LIN {X 0,Y 258.498,Z 368.712,A -85,B 0,C 180,E1 10982.882,E2 10982.882} C_VEL
LIN {X 0,Y 257.124,Z 367.282,A -85,B 0,C 180,E1 10976.432,E2 10976.432} C_VEL
LIN {X 0,Y 258.634,Z 368.161,A -85,B 0,C 180,E1 10970.206,E2 10970.206} C_VEL
LIN {X 0,Y 260.244,Z 369.538,A -85,B 0,C 180,E1 10967.35,E2 10967.35} C_VEL
LIN {X 0,Y 264.157,Z 374.05,A -85,B 0,C 180,E1 10962.601,E2 10962.601} C_VEL
LIN {X 0,Y 265.383,Z 375.444,A -85,B 0,C 180,E1 10961.436,E2 10961.436} C_VEL
LIN {X 0,Y 269.346,Z 380.009,A -85,B 0,C 180,E1 10958.209,E2 10958.209} C_VEL
LIN {X 0,Y 274.462,Z 386.667,A -85,B 0,C 180,E1 10954.771,E2 10954.771} C_VEL
LIN {X 0,Y 278.575,Z 392.041,A -85,B 0,C 180,E1 10952.418,E2 10952.418} C_VEL
LIN {X 0,Y 284.268,Z 399.8,A -85,B 0,C 180,E1 10949.569,E2 10949.569} C_VEL
LIN {X 0,Y 291.804,Z 410.986,A -85,B 0,C 180,E1 10946.283,E2 10946.283} C_VEL
LIN {X 0,Y 299.681,Z 423.896,A -85,B 0,C 180,E1 10943.269,E2 10943.269} C_VEL
LIN {X 0,Y 305.653,Z 435.016,A -85,B 0,C 180,E1 10941.187,E2 10941.187} C_VEL
LIN {X 0,Y 297.3,Z 573.705,A -85,B 0,C 180,E1 10938.161,E2 10938.161} C_VEL
LIN {X 0,Y 295.55,Z 593.68,A -85,B 0,C 180,E1 10937.44,E2 10937.44} C_VEL
LIN {X 0,Y 292.801,Z 612.599,A -85,B 0,C 180,E1 10936.45,E2 10936.45} C_VEL
LIN {X 0,Y 289.102,Z 631.006,A -85,B 0,C 180,E1 10935.151,E2 10935.151} C_VEL
LIN {X 0,Y 284.543,Z 648.768,A -85,B 0,C 180,E1 10933.528,E2 10933.528} C_VEL
LIN {X 0,Y 279.319,Z 665.496,A -85,B 0,C 180,E1 10931.592,E2 10931.592} C_VEL
LIN {X 0,Y 273.668,Z 681.017,A -85,B 0,C 180,E1 10929.336,E2 10929.336} C_VEL
LIN {X 0,Y 267.659,Z 695.529,A -85,B 0,C 180,E1 10926.703,E2 10926.703} C_VEL
LIN {X 0,Y 261.523,Z 708.893,A -85,B 0,C 180,E1 10923.666,E2 10923.666} C_VEL
LIN {X 0,Y 255.629,Z 720.676,A -85,B 0,C 180,E1 10920.302,E2 10920.302} C_VEL
LIN {X 0,Y 250.186,Z 730.94,A -85,B 0,C 180,E1 10916.589,E2 10916.589} C_VEL
LIN {X 0,Y 245.383,Z 739.687,A -85,B 0,C 180,E1 10912.52,E2 10912.52} C_VEL
LIN {X 0,Y 241.368,Z 746.89,A -85,B 0,C 180,E1 10908.1,E2 10908.1} C_VEL
LIN {X 0,Y 238.336,Z 752.477,A -85,B 0,C 180,E1 10903.34,E2 10903.34} C_VEL
LIN {X 0,Y 236.388,Z 756.219,A -85,B 0,C 180,E1 10898.513,E2 10898.513} C_VEL
LIN {X 0,Y 235.4,Z 758.256,A -85,B 0,C 180,E1 10893.653,E2 10893.653} C_VEL
LIN {X 0,Y 235.216,Z 758.676,A -85,B 0,C 180,E1 10888.782,E2 10888.782} C_VEL
LIN {X 0,Y 235.771,Z 757.501,A -85,B 0,C 180,E1 10883.914,E2 10883.914} C_VEL
LIN {X 0,Y 237.208,Z 754.67,A -85,B 0,C 180,E1 10879.066,E2 10879.066} C_VEL
LIN {X 0,Y 239.658,Z 750.072,A -85,B 0,C 180,E1 10874.266,E2 10874.266} C_VEL
LIN {X 0,Y 243.275,Z 743.544,A -85,B 0,C 180,E1 10869.553,E2 10869.553} C_VEL
LIN {X 0,Y 247.587,Z 735.82,A -85,B 0,C 180,E1 10865.421,E2 10865.421} C_VEL
LIN {X 0,Y 252.864,Z 726.09,A -85,B 0,C 180,E1 10861.417,E2 10861.417} C_VEL
LIN {X 0,Y 258.607,Z 715.007,A -85,B 0,C 180,E1 10857.858,E2 10857.858} C_VEL
LIN {X 0,Y 264.609,Z 702.544,A -85,B 0,C 180,E1 10854.682,E2 10854.682} C_VEL
LIN {X 0,Y 270.597,Z 688.893,A -85,B 0,C 180,E1 10851.899,E2 10851.899} C_VEL
LIN {X 0,Y 276.586,Z 673.604,A -85,B 0,C 180,E1 10849.407,E2 10849.407} C_VEL
LIN {X 0,Y 282.163,Z 657.139,A -85,B 0,C 180,E1 10847.268,E2 10847.268} C_VEL
LIN {X 0,Y 286.946,Z 640.408,A -85,B 0,C 180,E1 10845.544,E2 10845.544} C_VEL
LIN {X 0,Y 291.03,Z 622.739,A -85,B 0,C 180,E1 10844.109,E2 10844.109} C_VEL
LIN {X 0,Y 294.382,Z 603.565,A -85,B 0,C 180,E1 10842.926,E2 10842.926} C_VEL
LIN {X 0,Y 296.689,Z 583.8,A -85,B 0,C 180,E1 10842.051,E2 10842.051} C_VEL
LIN {X 0,Y 298.203,Z 559.266,A -85,B 0,C 180,E1 10841.365,E2 10841.365} C_VEL
LIN {X 0,Y 305.696,Z 434.6,A -85,B 0,C 180,E1 10838.662,E2 10838.662} C_VEL
LIN {X 0,Y 297.082,Z 419.319,A -85,B 0,C 180,E1 10835.609,E2 10835.609} C_VEL
LIN {X 0,Y 288.785,Z 406.306,A -85,B 0,C 180,E1 10832.281,E2 10832.281} C_VEL
LIN {X 0,Y 284.011,Z 399.335,A -85,B 0,C 180,E1 10830.122,E2 10830.122} C_VEL
LIN {X 0,Y 281.149,Z 396.523,A -85,B 0,C 180,E1 10828.78,E2 10828.78} C_VEL
LIN {X 0,Y 276.362,Z 394.63,A -85,B 0,C 180,E1 10826.484,E2 10826.484} C_VEL
LIN {X 0,Y 271.794,Z 392.718,A -85,B 0,C 180,E1 10823.976,E2 10823.976} C_VEL
LIN {X 0,Y 270.944,Z 391.928,A -85,B 0,C 180,E1 10823.434,E2 10823.434} C_VEL
LIN {X 0,Y 267.351,Z 387.273,A -85,B 0,C 180,E1 10820.812,E2 10820.812} C_VEL
LIN {X 0,Y 263.114,Z 382.029,A -85,B 0,C 180,E1 10817.015,E2 10817.015} C_VEL
LIN {X 0,Y 258.557,Z 376.707,A -85,B 0,C 180,E1 10810.923,E2 10810.923} C_VEL
LIN {X 0,Y 256.5,Z 375.483,A -85,B 0,C 180,E1 10804.696,E2 10804.696} C_VEL
LIN {X 0,Y 257.092,Z 376.28,A -85,B 0,C 180,E1 10798.886,E2 10798.886} C_VEL
LIN {X 0,Y 257.981,Z 377.437,A -85,B 0,C 180,E1 10796.556,E2 10796.556} C_VEL
LIN {X 0,Y 261.729,Z 382.457,A -85,B 0,C 180,E1 10790.878,E2 10790.878} C_VEL
LIN {X 0,Y 265.913,Z 388.376,A -85,B 0,C 180,E1 10786.741,E2 10786.741} C_VEL
LIN {X 0,Y 269.411,Z 393.338,A -85,B 0,C 180,E1 10784.005,E2 10784.005} C_VEL
LIN {X 0,Y 273.262,Z 398.777,A -85,B 0,C 180,E1 10781.438,E2 10781.438} C_VEL
LIN {X 0,Y 279.044,Z 407.526,A -85,B 0,C 180,E1 10778.121,E2 10778.121} C_VEL
LIN {X 0,Y 285.652,Z 417.93,A -85,B 0,C 180,E1 10774.887,E2 10774.887} C_VEL
LIN {X 0,Y 292.882,Z 430.603,A -85,B 0,C 180,E1 10771.783,E2 10771.783} C_VEL
LIN {X 0,Y 300.457,Z 445.23,A -85,B 0,C 180,E1 10768.865,E2 10768.865} C_VEL
LIN {X 0,Y 301.565,Z 447.913,A -85,B 0,C 180,E1 10768.445,E2 10768.445} C_VEL
LIN {X 0,Y 289.159,Z 619.599,A -85,B 0,C 180,E1 10764.411,E2 10764.411} C_VEL
LIN {X 0,Y 286.147,Z 641.14,A -85,B 0,C 180,E1 10763.637,E2 10763.637} C_VEL
LIN {X 0,Y 281.87,Z 661.827,A -85,B 0,C 180,E1 10762.613,E2 10762.613} C_VEL
LIN {X 0,Y 276.706,Z 681.385,A -85,B 0,C 180,E1 10761.304,E2 10761.304} C_VEL
LIN {X 0,Y 270.978,Z 699.735,A -85,B 0,C 180,E1 10759.689,E2 10759.689} C_VEL
LIN {X 0,Y 264.827,Z 717.159,A -85,B 0,C 180,E1 10757.73,E2 10757.73} C_VEL
LIN {X 0,Y 258.142,Z 734.335,A -85,B 0,C 180,E1 10755.294,E2 10755.294} C_VEL
LIN {X 0,Y 251.348,Z 750.591,A -85,B 0,C 180,E1 10752.396,E2 10752.396} C_VEL
LIN {X 0,Y 244.707,Z 765.827,A -85,B 0,C 180,E1 10748.992,E2 10748.992} C_VEL
LIN {X 0,Y 238.534,Z 779.922,A -85,B 0,C 180,E1 10745.047,E2 10745.047} C_VEL
LIN {X 0,Y 233.305,Z 792.414,A -85,B 0,C 180,E1 10740.662,E2 10740.662} C_VEL
LIN {X 0,Y 229.251,Z 803.286,A -85,B 0,C 180,E1 10735.857,E2 10735.857} C_VEL
LIN {X 0,Y 226.686,Z 812.077,A -85,B 0,C 180,E1 10730.932,E2 10730.932} C_VEL
LIN {X 0,Y 225.473,Z 818.98,A -85,B 0,C 180,E1 10725.958,E2 10725.958} C_VEL
LIN {X 0,Y 225.358,Z 824.09,A -85,B 0,C 180,E1 10720.998,E2 10720.998} C_VEL
LIN {X 0,Y 225.895,Z 827.071,A -85,B 0,C 180,E1 10716.608,E2 10716.608} C_VEL
LIN {X 0,Y 226.468,Z 828.64,A -85,B 0,C 180,E1 10712.53,E2 10712.53} C_VEL
LIN {X 0,Y 226.592,Z 828.825,A -85,B 0,C 180,E1 10708.989,E2 10708.989} C_VEL
LIN {X 0,Y 226.217,Z 827.996,A -85,B 0,C 180,E1 10705.437,E2 10705.437} C_VEL
LIN {X 0,Y 225.544,Z 825.443,A -85,B 0,C 180,E1 10700.817,E2 10700.817} C_VEL
LIN {X 0,Y 225.306,Z 821.337,A -85,B 0,C 180,E1 10696.135,E2 10696.135} C_VEL
LIN {X 0,Y 226.015,Z 815.194,A -85,B 0,C 180,E1 10691.16,E2 10691.16} C_VEL
LIN {X 0,Y 228.001,Z 807.19,A -85,B 0,C 180,E1 10686.207,E2 10686.207} C_VEL
LIN {X 0,Y 231.197,Z 797.77,A -85,B 0,C 180,E1 10681.595,E2 10681.595} C_VEL
LIN {X 0,Y 235.747,Z 786.348,A -85,B 0,C 180,E1 10677.115,E2 10677.115} C_VEL
LIN {X 0,Y 241.29,Z 773.485,A -85,B 0,C 180,E1 10673.07,E2 10673.07} C_VEL
LIN {X 0,Y 247.734,Z 758.735,A -85,B 0,C 180,E1 10669.355,E2 10669.355} C_VEL
LIN {X 0,Y 254.404,Z 743.211,A -85,B 0,C 180,E1 10666.236,E2 10666.236} C_VEL
LIN {X 0,Y 261.141,Z 726.599,A -85,B 0,C 180,E1 10663.565,E2 10663.565} C_VEL
LIN {X 0,Y 267.636,Z 709.13,A -85,B 0,C 180,E1 10661.332,E2 10661.332} C_VEL
LIN {X 0,Y 273.575,Z 691.374,A -85,B 0,C 180,E1 10659.544,E2 10659.544} C_VEL
LIN {X 0,Y 279.247,Z 671.79,A -85,B 0,C 180,E1 10658.029,E2 10658.029} C_VEL
LIN {X 0,Y 284.025,Z 651.634,A -85,B 0,C 180,E1 10656.866,E2 10656.866} C_VEL
LIN {X 0,Y 287.728,Z 630.265,A -85,B 0,C 180,E1 10655.959,E2 10655.959} C_VEL
LIN {X 0,Y 290.003,Z 608.45,A -85,B 0,C 180,E1 10655.313,E2 10655.313} C_VEL
LIN {X 0,Y 301.425,Z 447.468,A -85,B 0,C 180,E1 10651.552,E2 10651.552} C_VEL
LIN {X 0,Y 294.484,Z 433.716,A -85,B 0,C 180,E1 10648.935,E2 10648.935} C_VEL
LIN {X 0,Y 287.224,Z 420.756,A -85,B 0,C 180,E1 10645.904,E2 10645.904} C_VEL
LIN {X 0,Y 280.376,Z 409.547,A -85,B 0,C 180,E1 10642.652,E2 10642.652} C_VEL
LIN {X 0,Y 274.472,Z 400.605,A -85,B 0,C 180,E1 10639.415,E2 10639.415} C_VEL
LIN {X 0,Y 271.055,Z 395.721,A -85,B 0,C 180,E1 10637.274,E2 10637.274} C_VEL
LIN {X 0,Y 267.364,Z 390.484,A -85,B 0,C 180,E1 10634.621,E2 10634.621} C_VEL
LIN {X 0,Y 264.503,Z 386.557,A -85,B 0,C 180,E1 10632.221,E2 10632.221} C_VEL
LIN {X 0,Y 261.043,Z 381.597,A -85,B 0,C 180,E1 10628.591,E2 10628.591} C_VEL
LIN {X 0,Y 257.415,Z 376.588,A -85,B 0,C 180,E1 10622.671,E2 10622.671} C_VEL
LIN {X 0,Y 256.15,Z 375.222,A -85,B 0,C 180,E1 10616.419,E2 10616.419} C_VEL
LIN {X 0,Y 257.568,Z 376.056,A -85,B 0,C 180,E1 10610.391,E2 10610.391} C_VEL
LIN {X 0,Y 259.069,Z 377.366,A -85,B 0,C 180,E1 10607.631,E2 10607.631} C_VEL
LIN {X 0,Y 262.995,Z 381.948,A -85,B 0,C 180,E1 10602.749,E2 10602.749} C_VEL
LIN {X 0,Y 268.301,Z 388.521,A -85,B 0,C 180,E1 10598.177,E2 10598.177} C_VEL
LIN {X 0,Y 272.616,Z 394.185,A -85,B 0,C 180,E1 10595.226,E2 10595.226} C_VEL
LIN {X 0,Y 276.563,Z 399.467,A -85,B 0,C 180,E1 10592.901,E2 10592.901} C_VEL
LIN {X 0,Y 281.943,Z 406.999,A -85,B 0,C 180,E1 10590.115,E2 10590.115} C_VEL
LIN {X 0,Y 288.994,Z 417.776,A -85,B 0,C 180,E1 10586.921,E2 10586.921} C_VEL
LIN {X 0,Y 296.356,Z 430.137,A -85,B 0,C 180,E1 10583.992,E2 10583.992} C_VEL
LIN {X 0,Y 300.821,Z 438.681,A -85,B 0,C 180,E1 10582.35,E2 10582.35} C_VEL
LIN {X 0,Y 292.308,Z 574.377,A -85,B 0,C 180,E1 10579.369,E2 10579.369} C_VEL
LIN {X 0,Y 290.51,Z 594.197,A -85,B 0,C 180,E1 10578.652,E2 10578.652} C_VEL
LIN {X 0,Y 287.595,Z 613.573,A -85,B 0,C 180,E1 10577.634,E2 10577.634} C_VEL
LIN {X 0,Y 283.709,Z 632.181,A -85,B 0,C 180,E1 10576.31,E2 10576.31} C_VEL
LIN {X 0,Y 278.888,Z 650.216,A -85,B 0,C 180,E1 10574.642,E2 10574.642} C_VEL
LIN {X 0,Y 273.57,Z 666.596,A -85,B 0,C 180,E1 10572.724,E2 10572.724} C_VEL
LIN {X 0,Y 267.61,Z 682.332,A -85,B 0,C 180,E1 10570.408,E2 10570.408} C_VEL
LIN {X 0,Y 261.367,Z 696.808,A -85,B 0,C 180,E1 10567.739,E2 10567.739} C_VEL
LIN {X 0,Y 254.976,Z 710.147,A -85,B 0,C 180,E1 10564.652,E2 10564.652} C_VEL
LIN {X 0,Y 248.823,Z 721.912,A -85,B 0,C 180,E1 10561.222,E2 10561.222} C_VEL
LIN {X 0,Y 243.121,Z 732.163,A -85,B 0,C 180,E1 10557.426,E2 10557.426} C_VEL
LIN {X 0,Y 238.075,Z 740.901,A -85,B 0,C 180,E1 10553.251,E2 10553.251} C_VEL
LIN {X 0,Y 233.84,Z 748.099,A -85,B 0,C 180,E1 10548.704,E2 10548.704} C_VEL
LIN {X 0,Y 230.628,Z 753.683,A -85,B 0,C 180,E1 10543.794,E2 10543.794} C_VEL
LIN {X 0,Y 228.557,Z 757.423,A -85,B 0,C 180,E1 10538.807,E2 10538.807} C_VEL
LIN {X 0,Y 227.505,Z 759.458,A -85,B 0,C 180,E1 10533.78,E2 10533.78} C_VEL
LIN {X 0,Y 227.308,Z 759.877,A -85,B 0,C 180,E1 10528.74,E2 10528.74} C_VEL
LIN {X 0,Y 227.901,Z 758.703,A -85,B 0,C 180,E1 10523.703,E2 10523.703} C_VEL
LIN {X 0,Y 229.437,Z 755.864,A -85,B 0,C 180,E1 10518.676,E2 10518.676} C_VEL
LIN {X 0,Y 232.031,Z 751.28,A -85,B 0,C 180,E1 10513.735,E2 10513.735} C_VEL
LIN {X 0,Y 235.857,Z 744.755,A -85,B 0,C 180,E1 10508.88,E2 10508.88} C_VEL
LIN {X 0,Y 240.395,Z 737.036,A -85,B 0,C 180,E1 10504.635,E2 10504.635} C_VEL
LIN {X 0,Y 245.933,Z 727.313,A -85,B 0,C 180,E1 10500.533,E2 10500.533} C_VEL
LIN {X 0,Y 251.704,Z 716.687,A -85,B 0,C 180,E1 10497.03,E2 10497.03} C_VEL
LIN {X 0,Y 258.196,Z 703.801,A -85,B 0,C 180,E1 10493.667,E2 10493.667} C_VEL
LIN {X 0,Y 264.573,Z 689.844,A -85,B 0,C 180,E1 10490.781,E2 10490.781} C_VEL
LIN {X 0,Y 270.644,Z 674.935,A -85,B 0,C 180,E1 10488.32,E2 10488.32} C_VEL
LIN {X 0,Y 276.427,Z 658.533,A -85,B 0,C 180,E1 10486.16,E2 10486.16} C_VEL
LIN {X 0,Y 281.647,Z 640.917,A -85,B 0,C 180,E1 10484.331,E2 10484.331} C_VEL
LIN {X 0,Y 285.882,Z 623.12,A -85,B 0,C 180,E1 10482.887,E2 10482.887} C_VEL
LIN {X 0,Y 289.324,Z 603.974,A -85,B 0,C 180,E1 10481.708,E2 10481.708} C_VEL
LIN {X 0,Y 291.689,Z 584.308,A -85,B 0,C 180,E1 10480.838,E2 10480.838} C_VEL
LIN {X 0,Y 293.267,Z 559.696,A -85,B 0,C 180,E1 10480.148,E2 10480.148} C_VEL
LIN {X 0,Y 300.922,Z 438.413,A -85,B 0,C 180,E1 10477.513,E2 10477.513} C_VEL
LIN {X 0,Y 293.599,Z 425.217,A -85,B 0,C 180,E1 10474.78,E2 10474.78} C_VEL
LIN {X 0,Y 285.958,Z 412.916,A -85,B 0,C 180,E1 10471.575,E2 10471.575} C_VEL
LIN {X 0,Y 278.692,Z 402.195,A -85,B 0,C 180,E1 10468.034,E2 10468.034} C_VEL
LIN {X 0,Y 274.332,Z 396.407,A -85,B 0,C 180,E1 10465.589,E2 10465.589} C_VEL
LIN {X 0,Y 271.016,Z 392.007,A -85,B 0,C 180,E1 10463.481,E2 10463.481} C_VEL
LIN {X 0,Y 270.944,Z 391.928,A -85,B 0,C 180,E1 10463.434,E2 10463.434} C_VEL
LIN {X 0,Y 268.454,Z 390.258,A -85,B 0,C 180,E1 10461.789,E2 10461.789} C_VEL
LIN {X 0,Y 261.646,Z 389.615,A -85,B 0,C 180,E1 10456.543,E2 10456.543} C_VEL
LIN {X 0,Y 261.183,Z 389.307,A -85,B 0,C 180,E1 10456.067,E2 10456.067} C_VEL
LIN {X 0,Y 257.474,Z 384.599,A -85,B 0,C 180,E1 10450.743,E2 10450.743} C_VEL
LIN {X 0,Y 255.529,Z 383.424,A -85,B 0,C 180,E1 10444.714,E2 10444.714} C_VEL
LIN {X 0,Y 256.047,Z 384.17,A -85,B 0,C 180,E1 10439.105,E2 10439.105} C_VEL
LIN {X 0,Y 256.846,Z 385.226,A -85,B 0,C 180,E1 10436.876,E2 10436.876} C_VEL
LIN {X 0,Y 260.346,Z 390.15,A -85,B 0,C 180,E1 10431.275,E2 10431.275} C_VEL
LIN {X 0,Y 264.395,Z 396.089,A -85,B 0,C 180,E1 10427.108,E2 10427.108} C_VEL
LIN {X 0,Y 267.601,Z 400.785,A -85,B 0,C 180,E1 10424.506,E2 10424.506} C_VEL
LIN {X 0,Y 271.269,Z 406.134,A -85,B 0,C 180,E1 10421.965,E2 10421.965} C_VEL
LIN {X 0,Y 276.735,Z 414.653,A -85,B 0,C 180,E1 10418.709,E2 10418.709} C_VEL
LIN {X 0,Y 282.895,Z 424.631,A -85,B 0,C 180,E1 10415.574,E2 10415.574} C_VEL
LIN {X 0,Y 289.751,Z 437.071,A -85,B 0,C 180,E1 10412.486,E2 10412.486} C_VEL
LIN {X 0,Y 296.819,Z 451.107,A -85,B 0,C 180,E1 10409.642,E2 10409.642} C_VEL
LIN {X 0,Y 284.291,Z 618.719,A -85,B 0,C 180,E1 10405.694,E2 10405.694} C_VEL
LIN {X 0,Y 281.194,Z 640.264,A -85,B 0,C 180,E1 10404.92,E2 10404.92} C_VEL
LIN {X 0,Y 276.844,Z 660.774,A -85,B 0,C 180,E1 10403.909,E2 10403.909} C_VEL
LIN {X 0,Y 271.301,Z 681.09,A -85,B 0,C 180,E1 10402.549,E2 10402.549} C_VEL
LIN {X 0,Y 265.037,Z 700.385,A -85,B 0,C 180,E1 10400.826,E2 10400.826} C_VEL
LIN {X 0,Y 258.217,Z 718.776,A -85,B 0,C 180,E1 10398.692,E2 10398.692} C_VEL
LIN {X 0,Y 251.075,Z 736.136,A -85,B 0,C 180,E1 10396.118,E2 10396.118} C_VEL
LIN {X 0,Y 244.095,Z 751.924,A -85,B 0,C 180,E1 10393.16,E2 10393.16} C_VEL
LIN {X 0,Y 237.463,Z 766.313,A -85,B 0,C 180,E1 10389.791,E2 10389.791} C_VEL
LIN {X 0,Y 231.406,Z 779.378,A -85,B 0,C 180,E1 10385.988,E2 10385.988} C_VEL
LIN {X 0,Y 225.893,Z 791.752,A -85,B 0,C 180,E1 10381.485,E2 10381.485} C_VEL
LIN {X 0,Y 221.593,Z 802.519,A -85,B 0,C 180,E1 10376.531,E2 10376.531} C_VEL
LIN {X 0,Y 218.849,Z 811.216,A -85,B 0,C 180,E1 10371.437,E2 10371.437} C_VEL
LIN {X 0,Y 217.501,Z 818.328,A -85,B 0,C 180,E1 10366.01,E2 10366.01} C_VEL
LIN {X 0,Y 217.416,Z 823.253,A -85,B 0,C 180,E1 10360.868,E2 10360.868} C_VEL
LIN {X 0,Y 218,Z 826.132,A -85,B 0,C 180,E1 10356.319,E2 10356.319} C_VEL
LIN {X 0,Y 218.599,Z 827.503,A -85,B 0,C 180,E1 10352.097,E2 10352.097} C_VEL
LIN {X 0,Y 218.662,Z 827.594,A -85,B 0,C 180,E1 10348.69,E2 10348.69} C_VEL
LIN {X 0,Y 218.175,Z 826.603,A -85,B 0,C 180,E1 10344.741,E2 10344.741} C_VEL
LIN {X 0,Y 217.525,Z 824.016,A -85,B 0,C 180,E1 10340.208,E2 10340.208} C_VEL
LIN {X 0,Y 217.399,Z 819.492,A -85,B 0,C 180,E1 10335.075,E2 10335.075} C_VEL
LIN {X 0,Y 218.362,Z 813.188,A -85,B 0,C 180,E1 10329.915,E2 10329.915} C_VEL
LIN {X 0,Y 220.725,Z 804.999,A -85,B 0,C 180,E1 10324.799,E2 10324.799} C_VEL
LIN {X 0,Y 224.747,Z 794.465,A -85,B 0,C 180,E1 10319.662,E2 10319.662} C_VEL
LIN {X 0,Y 230.05,Z 782.292,A -85,B 0,C 180,E1 10314.992,E2 10314.992} C_VEL
LIN {X 0,Y 236.245,Z 768.859,A -85,B 0,C 180,E1 10310.906,E2 10310.906} C_VEL
LIN {X 0,Y 243.147,Z 753.856,A -85,B 0,C 180,E1 10307.274,E2 10307.274} C_VEL
LIN {X 0,Y 250.279,Z 737.764,A -85,B 0,C 180,E1 10304.186,E2 10304.186} C_VEL
LIN {X 0,Y 257.346,Z 720.677,A -85,B 0,C 180,E1 10301.592,E2 10301.592} C_VEL
LIN {X 0,Y 263.764,Z 703.556,A -85,B 0,C 180,E1 10299.538,E2 10299.538} C_VEL
LIN {X 0,Y 269.728,Z 685.704,A -85,B 0,C 180,E1 10297.857,E2 10297.857} C_VEL
LIN {X 0,Y 275.313,Z 666.188,A -85,B 0,C 180,E1 10296.447,E2 10296.447} C_VEL
LIN {X 0,Y 280.038,Z 645.527,A -85,B 0,C 180,E1 10295.34,E2 10295.34} C_VEL
LIN {X 0,Y 283.464,Z 624.268,A -85,B 0,C 180,E1 10294.508,E2 10294.508} C_VEL
LIN {X 0,Y 285.834,Z 598.19,A -85,B 0,C 180,E1 10293.805,E2 10293.805} C_VEL
LIN {X 0,Y 296.611,Z 450.834,A -85,B 0,C 180,E1 10290.346,E2 10290.346} C_VEL
LIN {X 0,Y 289.027,Z 435.767,A -85,B 0,C 180,E1 10287.282,E2 10287.282} C_VEL
LIN {X 0,Y 282.139,Z 423.569,A -85,B 0,C 180,E1 10284.161,E2 10284.161} C_VEL
LIN {X 0,Y 276.319,Z 414.042,A -85,B 0,C 180,E1 10281.158,E2 10281.158} C_VEL
LIN {X 0,Y 270.063,Z 404.188,A -85,B 0,C 180,E1 10277.339,E2 10277.339} C_VEL
LIN {X 0,Y 265.445,Z 397.664,A -85,B 0,C 180,E1 10273.949,E2 10273.949} C_VEL
LIN {X 0,Y 262.933,Z 394.104,A -85,B 0,C 180,E1 10271.738,E2 10271.738} C_VEL
LIN {X 0,Y 259.698,Z 389.302,A -85,B 0,C 180,E1 10268.189,E2 10268.189} C_VEL
LIN {X 0,Y 256.345,Z 384.467,A -85,B 0,C 180,E1 10262.459,E2 10262.459} C_VEL
LIN {X 0,Y 255.184,Z 383.158,A -85,B 0,C 180,E1 10256.18,E2 10256.18} C_VEL
LIN {X 0,Y 256.707,Z 384.087,A -85,B 0,C 180,E1 10250.132,E2 10250.132} C_VEL
LIN {X 0,Y 257.898,Z 385.192,A -85,B 0,C 180,E1 10247.915,E2 10247.915} C_VEL
LIN {X 0,Y 262.35,Z 390.573,A -85,B 0,C 180,E1 10242.362,E2 10242.362} C_VEL
LIN {X 0,Y 266.721,Z 396.22,A -85,B 0,C 180,E1 10238.561,E2 10238.561} C_VEL
LIN {X 0,Y 270.799,Z 401.697,A -85,B 0,C 180,E1 10235.689,E2 10235.689} C_VEL
LIN {X 0,Y 274.657,Z 407.011,A -85,B 0,C 180,E1 10233.341,E2 10233.341} C_VEL
LIN {X 0,Y 279.64,Z 414.192,A -85,B 0,C 180,E1 10230.669,E2 10230.669} C_VEL
LIN {X 0,Y 286.222,Z 424.561,A -85,B 0,C 180,E1 10227.573,E2 10227.573} C_VEL
LIN {X 0,Y 293.136,Z 436.486,A -85,B 0,C 180,E1 10224.709,E2 10224.709} C_VEL
LIN {X 0,Y 296.121,Z 442.35,A -85,B 0,C 180,E1 10223.551,E2 10223.551} C_VEL
LIN {X 0,Y 287.45,Z 575.037,A -85,B 0,C 180,E1 10220.618,E2 10220.618} C_VEL
LIN {X 0,Y 285.615,Z 594.636,A -85,B 0,C 180,E1 10219.909,E2 10219.909} C_VEL
LIN {X 0,Y 282.763,Z 613.24,A -85,B 0,C 180,E1 10218.941,E2 10218.941} C_VEL
LIN {X 0,Y 278.956,Z 631.262,A -85,B 0,C 180,E1 10217.684,E2 10217.684} C_VEL
LIN {X 0,Y 274.431,Z 648.157,A -85,B 0,C 180,E1 10216.168,E2 10216.168} C_VEL
LIN {X 0,Y 269.082,Z 664.6,A -85,B 0,C 180,E1 10214.311,E2 10214.311} C_VEL
LIN {X 0,Y 262.908,Z 680.715,A -85,B 0,C 180,E1 10212.015,E2 10212.015} C_VEL
LIN {X 0,Y 256.578,Z 695.169,A -85,B 0,C 180,E1 10209.433,E2 10209.433} C_VEL
LIN {X 0,Y 249.799,Z 708.983,A -85,B 0,C 180,E1 10206.326,E2 10206.326} C_VEL
LIN {X 0,Y 243.239,Z 721.158,A -85,B 0,C 180,E1 10202.86,E2 10202.86} C_VEL
LIN {X 0,Y 237.107,Z 731.773,A -85,B 0,C 180,E1 10199.008,E2 10199.008} C_VEL
LIN {X 0,Y 231.628,Z 740.837,A -85,B 0,C 180,E1 10194.753,E2 10194.753} C_VEL
LIN {X 0,Y 226.97,Z 748.334,A -85,B 0,C 180,E1 10190.096,E2 10190.096} C_VEL
LIN {X 0,Y 223.517,Z 753.966,A -85,B 0,C 180,E1 10185.303,E2 10185.303} C_VEL
LIN {X 0,Y 221.088,Z 758.053,A -85,B 0,C 180,E1 10180.158,E2 10180.158} C_VEL
LIN {X 0,Y 219.761,Z 760.419,A -85,B 0,C 180,E1 10174.959,E2 10174.959} C_VEL
LIN {X 0,Y 219.383,Z 761.161,A -85,B 0,C 180,E1 10169.739,E2 10169.739} C_VEL
LIN {X 0,Y 219.84,Z 760.314,A -85,B 0,C 180,E1 10164.52,E2 10164.52} C_VEL
LIN {X 0,Y 221.255,Z 757.829,A -85,B 0,C 180,E1 10159.323,E2 10159.323} C_VEL
LIN {X 0,Y 223.781,Z 753.598,A -85,B 0,C 180,E1 10154.184,E2 10154.184} C_VEL
LIN {X 0,Y 227.562,Z 747.464,A -85,B 0,C 180,E1 10149.152,E2 10149.152} C_VEL
LIN {X 0,Y 232.39,Z 739.694,A -85,B 0,C 180,E1 10144.517,E2 10144.517} C_VEL
LIN {X 0,Y 237.688,Z 730.931,A -85,B 0,C 180,E1 10140.518,E2 10140.518} C_VEL
LIN {X 0,Y 243.916,Z 720.117,A -85,B 0,C 180,E1 10136.683,E2 10136.683} C_VEL
LIN {X 0,Y 250.552,Z 707.71,A -85,B 0,C 180,E1 10133.232,E2 10133.232} C_VEL
LIN {X 0,Y 257.163,Z 694.13,A -85,B 0,C 180,E1 10130.241,E2 10130.241} C_VEL
LIN {X 0,Y 263.541,Z 679.487,A -85,B 0,C 180,E1 10127.67,E2 10127.67} C_VEL
LIN {X 0,Y 269.486,Z 663.857,A -85,B 0,C 180,E1 10125.475,E2 10125.475} C_VEL
LIN {X 0,Y 275.126,Z 646.327,A -85,B 0,C 180,E1 10123.531,E2 10123.531} C_VEL
LIN {X 0,Y 279.779,Z 628.546,A -85,B 0,C 180,E1 10121.985,E2 10121.985} C_VEL
LIN {X 0,Y 283.603,Z 609.532,A -85,B 0,C 180,E1 10120.724,E2 10120.724} C_VEL
LIN {X 0,Y 286.324,Z 590.113,A -85,B 0,C 180,E1 10119.782,E2 10119.782} C_VEL
LIN {X 0,Y 287.927,Z 569.881,A -85,B 0,C 180,E1 10119.124,E2 10119.124} C_VEL
LIN {X 0,Y 296.194,Z 442.051,A -85,B 0,C 180,E1 10116.301,E2 10116.301} C_VEL
LIN {X 0,Y 289.578,Z 430.115,A -85,B 0,C 180,E1 10113.685,E2 10113.685} C_VEL
LIN {X 0,Y 282.871,Z 419.072,A -85,B 0,C 180,E1 10110.715,E2 10110.715} C_VEL
LIN {X 0,Y 276.297,Z 409.138,A -85,B 0,C 180,E1 10107.361,E2 10107.361} C_VEL
LIN {X 0,Y 272.076,Z 403.378,A -85,B 0,C 180,E1 10104.884,E2 10104.884} C_VEL
LIN {X 0,Y 269.172,Z 399.4,A -85,B 0,C 180,E1 10102.957,E2 10102.957} C_VEL
LIN {X 0,Y 265.748,Z 394.853,A -85,B 0,C 180,E1 10100.367,E2 10100.367} C_VEL
LIN {X 0,Y 261.743,Z 389.755,A -85,B 0,C 180,E1 10096.649,E2 10096.649} C_VEL
LIN {X 0,Y 261.183,Z 389.307,A -85,B 0,C 180,E1 10096.067,E2 10096.067} C_VEL
LIN {X 0,Y 259.511,Z 388.941,A -85,B 0,C 180,E1 10094.267,E2 10094.267} C_VEL
LIN {X 0,Y 255.675,Z 391.866,A -85,B 0,C 180,E1 10088.992,E2 10088.992} C_VEL
LIN {X 0,Y 255.366,Z 391.84,A -85,B 0,C 180,E1 10088.238,E2 10088.238} C_VEL
LIN {X 0,Y 254.495,Z 391.444,A -85,B 0,C 180,E1 10082.477,E2 10082.477} C_VEL
LIN {X 0,Y 255.648,Z 392.802,A -85,B 0,C 180,E1 10077.423,E2 10077.423} C_VEL
LIN {X 0,Y 259,Z 397.844,A -85,B 0,C 180,E1 10071.677,E2 10071.677} C_VEL
LIN {X 0,Y 262.804,Z 403.617,A -85,B 0,C 180,E1 10067.587,E2 10067.587} C_VEL
LIN {X 0,Y 265.841,Z 408.235,A -85,B 0,C 180,E1 10065.015,E2 10065.015} C_VEL
LIN {X 0,Y 269.328,Z 413.494,A -85,B 0,C 180,E1 10062.5,E2 10062.5} C_VEL
LIN {X 0,Y 274.561,Z 421.92,A -85,B 0,C 180,E1 10059.259,E2 10059.259} C_VEL
LIN {X 0,Y 280.356,Z 431.69,A -85,B 0,C 180,E1 10056.179,E2 10056.179} C_VEL
LIN {X 0,Y 286.717,Z 443.639,A -85,B 0,C 180,E1 10053.182,E2 10053.182} C_VEL
LIN {X 0,Y 292.164,Z 454.872,A -85,B 0,C 180,E1 10050.862,E2 10050.862} C_VEL
LIN {X 0,Y 279.571,Z 617.839,A -85,B 0,C 180,E1 10047.02,E2 10047.02} C_VEL
LIN {X 0,Y 276.387,Z 639.389,A -85,B 0,C 180,E1 10046.249,E2 10046.249} C_VEL
LIN {X 0,Y 271.967,Z 659.718,A -85,B 0,C 180,E1 10045.25,E2 10045.25} C_VEL
LIN {X 0,Y 266.475,Z 679.3,A -85,B 0,C 180,E1 10043.956,E2 10043.956} C_VEL
LIN {X 0,Y 260.254,Z 697.966,A -85,B 0,C 180,E1 10042.316,E2 10042.316} C_VEL
LIN {X 0,Y 253.455,Z 715.829,A -85,B 0,C 180,E1 10040.285,E2 10040.285} C_VEL
LIN {X 0,Y 246.249,Z 732.855,A -85,B 0,C 180,E1 10037.816,E2 10037.816} C_VEL
LIN {X 0,Y 238.937,Z 748.793,A -85,B 0,C 180,E1 10034.894,E2 10034.894} C_VEL
LIN {X 0,Y 232.005,Z 763.19,A -85,B 0,C 180,E1 10031.58,E2 10031.58} C_VEL
LIN {X 0,Y 225.452,Z 776.562,A -85,B 0,C 180,E1 10027.734,E2 10027.734} C_VEL
LIN {X 0,Y 219.696,Z 788.576,A -85,B 0,C 180,E1 10023.413,E2 10023.413} C_VEL
LIN {X 0,Y 215.016,Z 799.192,A -85,B 0,C 180,E1 10018.617,E2 10018.617} C_VEL
LIN {X 0,Y 211.658,Z 808.331,A -85,B 0,C 180,E1 10013.378,E2 10013.378} C_VEL
LIN {X 0,Y 209.773,Z 815.863,A -85,B 0,C 180,E1 10007.76,E2 10007.76} C_VEL
LIN {X 0,Y 209.373,Z 821.127,A -85,B 0,C 180,E1 10002.409,E2 10002.409} C_VEL
LIN {X 0,Y 209.898,Z 824.487,A -85,B 0,C 180,E1 9997.389,E2 9997.389} C_VEL
LIN {X 0,Y 210.577,Z 826.182,A -85,B 0,C 180,E1 9992.994,E2 9992.994} C_VEL
LIN {X 0,Y 210.778,Z 826.448,A -85,B 0,C 180,E1 9989.185,E2 9989.185} C_VEL
LIN {X 0,Y 210.346,Z 825.659,A -85,B 0,C 180,E1 9985.365,E2 9985.365} C_VEL
LIN {X 0,Y 209.626,Z 823.367,A -85,B 0,C 180,E1 9980.667,E2 9980.667} C_VEL
LIN {X 0,Y 209.41,Z 819.115,A -85,B 0,C 180,E1 9975.342,E2 9975.342} C_VEL
LIN {X 0,Y 210.328,Z 813.021,A -85,B 0,C 180,E1 9969.985,E2 9969.985} C_VEL
LIN {X 0,Y 212.703,Z 805.097,A -85,B 0,C 180,E1 9964.675,E2 9964.675} C_VEL
LIN {X 0,Y 216.415,Z 795.766,A -85,B 0,C 180,E1 9959.763,E2 9959.763} C_VEL
LIN {X 0,Y 221.57,Z 784.454,A -85,B 0,C 180,E1 9955.034,E2 9955.034} C_VEL
LIN {X 0,Y 227.784,Z 771.682,A -85,B 0,C 180,E1 9950.797,E2 9950.797} C_VEL
LIN {X 0,Y 234.715,Z 757.432,A -85,B 0,C 180,E1 9947.034,E2 9947.034} C_VEL
LIN {X 0,Y 241.925,Z 742.23,A -85,B 0,C 180,E1 9943.848,E2 9943.848} C_VEL
LIN {X 0,Y 249.028,Z 726.281,A -85,B 0,C 180,E1 9941.182,E2 9941.182} C_VEL
LIN {X 0,Y 256.166,Z 708.698,A -85,B 0,C 180,E1 9938.862,E2 9938.862} C_VEL
LIN {X 0,Y 262.822,Z 690.255,A -85,B 0,C 180,E1 9936.976,E2 9936.976} C_VEL
LIN {X 0,Y 268.896,Z 670.685,A -85,B 0,C 180,E1 9935.455,E2 9935.455} C_VEL
LIN {X 0,Y 274.036,Z 650.32,A -85,B 0,C 180,E1 9934.276,E2 9934.276} C_VEL
LIN {X 0,Y 277.885,Z 629.512,A -85,B 0,C 180,E1 9933.388,E2 9933.388} C_VEL
LIN {X 0,Y 280.301,Z 608.505,A -85,B 0,C 180,E1 9932.751,E2 9932.751} C_VEL
LIN {X 0,Y 291.986,Z 454.521,A -85,B 0,C 180,E1 9929.131,E2 9929.131} C_VEL
LIN {X 0,Y 285.192,Z 440.776,A -85,B 0,C 180,E1 9926.215,E2 9926.215} C_VEL
LIN {X 0,Y 278.763,Z 429.163,A -85,B 0,C 180,E1 9923.125,E2 9923.125} C_VEL
LIN {X 0,Y 272.711,Z 418.917,A -85,B 0,C 180,E1 9919.768,E2 9919.768} C_VEL
LIN {X 0,Y 267.395,Z 410.591,A -85,B 0,C 180,E1 9916.286,E2 9916.286} C_VEL
LIN {X 0,Y 263.81,Z 405.188,A -85,B 0,C 180,E1 9913.479,E2 9913.479} C_VEL
LIN {X 0,Y 261.382,Z 401.648,A -85,B 0,C 180,E1 9911.249,E2 9911.249} C_VEL
LIN {X 0,Y 258.367,Z 397.007,A -85,B 0,C 180,E1 9907.784,E2 9907.784} C_VEL
LIN {X 0,Y 255.278,Z 392.346,A -85,B 0,C 180,E1 9902.244,E2 9902.244} C_VEL
LIN {X 0,Y 254.211,Z 391.099,A -85,B 0,C 180,E1 9896.166,E2 9896.166} C_VEL
LIN {X 0,Y 255.704,Z 392.024,A -85,B 0,C 180,E1 9890.18,E2 9890.18} C_VEL
LIN {X 0,Y 256.735,Z 393.017,A -85,B 0,C 180,E1 9888.201,E2 9888.201} C_VEL
LIN {X 0,Y 260.957,Z 398.313,A -85,B 0,C 180,E1 9882.725,E2 9882.725} C_VEL
LIN {X 0,Y 265.1,Z 403.811,A -85,B 0,C 180,E1 9879.003,E2 9879.003} C_VEL
LIN {X 0,Y 268.996,Z 409.205,A -85,B 0,C 180,E1 9876.157,E2 9876.157} C_VEL
LIN {X 0,Y 272.766,Z 414.545,A -85,B 0,C 180,E1 9873.787,E2 9873.787} C_VEL
LIN {X 0,Y 278.112,Z 422.513,A -85,B 0,C 180,E1 9870.846,E2 9870.846} C_VEL
LIN {X 0,Y 284.616,Z 433.283,A -85,B 0,C 180,E1 9867.725,E2 9867.725} C_VEL
LIN {X 0,Y 290.508,Z 443.893,A -85,B 0,C 180,E1 9865.216,E2 9865.216} C_VEL
LIN {X 0,Y 291.54,Z 446.205,A -85,B 0,C 180,E1 9864.786,E2 9864.786} C_VEL
LIN {X 0,Y 282.742,Z 575.597,A -85,B 0,C 180,E1 9861.913,E2 9861.913} C_VEL
LIN {X 0,Y 280.872,Z 595,A -85,B 0,C 180,E1 9861.213,E2 9861.213} C_VEL
LIN {X 0,Y 277.943,Z 613.625,A -85,B 0,C 180,E1 9860.249,E2 9860.249} C_VEL
LIN {X 0,Y 274.124,Z 631.298,A -85,B 0,C 180,E1 9859.026,E2 9859.026} C_VEL
LIN {X 0,Y 269.323,Z 648.727,A -85,B 0,C 180,E1 9857.469,E2 9857.469} C_VEL
LIN {X 0,Y 263.643,Z 665.595,A -85,B 0,C 180,E1 9855.557,E2 9855.557} C_VEL
LIN {X 0,Y 257.362,Z 681.441,A -85,B 0,C 180,E1 9853.29,E2 9853.29} C_VEL
LIN {X 0,Y 250.524,Z 696.445,A -85,B 0,C 180,E1 9850.581,E2 9850.581} C_VEL
LIN {X 0,Y 243.924,Z 709.41,A -85,B 0,C 180,E1 9847.643,E2 9847.643} C_VEL
LIN {X 0,Y 237.034,Z 721.716,A -85,B 0,C 180,E1 9844.125,E2 9844.125} C_VEL
LIN {X 0,Y 230.56,Z 732.446,A -85,B 0,C 180,E1 9840.201,E2 9840.201} C_VEL
LIN {X 0,Y 224.744,Z 741.619,A -85,B 0,C 180,E1 9835.848,E2 9835.848} C_VEL
LIN {X 0,Y 219.767,Z 749.217,A -85,B 0,C 180,E1 9831.064,E2 9831.064} C_VEL
LIN {X 0,Y 215.877,Z 755.172,A -85,B 0,C 180,E1 9825.858,E2 9825.858} C_VEL
LIN {X 0,Y 213.295,Z 759.256,A -85,B 0,C 180,E1 9820.534,E2 9820.534} C_VEL
LIN {X 0,Y 211.878,Z 761.621,A -85,B 0,C 180,E1 9815.144,E2 9815.144} C_VEL
LIN {X 0,Y 211.474,Z 762.363,A -85,B 0,C 180,E1 9809.729,E2 9809.729} C_VEL
LIN {X 0,Y 211.963,Z 761.516,A -85,B 0,C 180,E1 9804.315,E2 9804.315} C_VEL
LIN {X 0,Y 213.473,Z 759.033,A -85,B 0,C 180,E1 9798.929,E2 9798.929} C_VEL
LIN {X 0,Y 216.16,Z 754.805,A -85,B 0,C 180,E1 9793.611,E2 9793.611} C_VEL
LIN {X 0,Y 220.164,Z 748.675,A -85,B 0,C 180,E1 9788.417,E2 9788.417} C_VEL
LIN {X 0,Y 225.254,Z 740.91,A -85,B 0,C 180,E1 9783.649,E2 9783.649} C_VEL
LIN {X 0,Y 230.836,Z 732.13,A -85,B 0,C 180,E1 9779.539,E2 9779.539} C_VEL
LIN {X 0,Y 237.338,Z 721.355,A -85,B 0,C 180,E1 9775.633,E2 9775.633} C_VEL
LIN {X 0,Y 244.262,Z 708.968,A -85,B 0,C 180,E1 9772.121,E2 9772.121} C_VEL
LIN {X 0,Y 251.141,Z 695.418,A -85,B 0,C 180,E1 9769.088,E2 9769.088} C_VEL
LIN {X 0,Y 257.684,Z 681.008,A -85,B 0,C 180,E1 9766.519,E2 9766.519} C_VEL
LIN {X 0,Y 263.925,Z 665.23,A -85,B 0,C 180,E1 9764.276,E2 9764.276} C_VEL
LIN {X 0,Y 269.696,Z 648.035,A -85,B 0,C 180,E1 9762.342,E2 9762.342} C_VEL
LIN {X 0,Y 274.583,Z 630.145,A -85,B 0,C 180,E1 9760.766,E2 9760.766} C_VEL
LIN {X 0,Y 278.565,Z 611.282,A -85,B 0,C 180,E1 9759.495,E2 9759.495} C_VEL
LIN {X 0,Y 281.476,Z 591.614,A -85,B 0,C 180,E1 9758.524,E2 9758.524} C_VEL
LIN {X 0,Y 283.188,Z 571.365,A -85,B 0,C 180,E1 9757.853,E2 9757.853} C_VEL
LIN {X 0,Y 291.6,Z 445.773,A -85,B 0,C 180,E1 9755.054,E2 9755.054} C_VEL
LIN {X 0,Y 285.244,Z 434.181,A -85,B 0,C 180,E1 9752.369,E2 9752.369} C_VEL
LIN {X 0,Y 278.341,Z 422.75,A -85,B 0,C 180,E1 9749.068,E2 9749.068} C_VEL
LIN {X 0,Y 272.996,Z 414.791,A -85,B 0,C 180,E1 9746.131,E2 9746.131} C_VEL
LIN {X 0,Y 269.694,Z 410.128,A -85,B 0,C 180,E1 9744.068,E2 9744.068} C_VEL
LIN {X 0,Y 267.051,Z 406.445,A -85,B 0,C 180,E1 9742.22,E2 9742.22} C_VEL
LIN {X 0,Y 264.021,Z 402.301,A -85,B 0,C 180,E1 9739.813,E2 9739.813} C_VEL
LIN {X 0,Y 260.323,Z 397.438,A -85,B 0,C 180,E1 9736.223,E2 9736.223} C_VEL
LIN {X 0,Y 256.394,Z 392.491,A -85,B 0,C 180,E1 9730.562,E2 9730.562} C_VEL
LIN {X 0,Y 255.366,Z 391.84,A -85,B 0,C 180,E1 9728.238,E2 9728.238} C_VEL
LIN {X 0,Y 254.732,Z 392.537,A -85,B 0,C 180,E1 9726.507,E2 9726.507} C_VEL
LIN {X 0,Y 253.646,Z 399.134,A -85,B 0,C 180,E1 9721.54,E2 9721.54} C_VEL
LIN {X 0,Y 253.773,Z 399.758,A -85,B 0,C 180,E1 9720.41,E2 9720.41} C_VEL
LIN {X 0,Y 254.615,Z 400.805,A -85,B 0,C 180,E1 9717.525,E2 9717.525} C_VEL
LIN {X 0,Y 257.746,Z 405.701,A -85,B 0,C 180,E1 9711.973,E2 9711.973} C_VEL
LIN {X 0,Y 261.341,Z 411.329,A -85,B 0,C 180,E1 9707.965,E2 9707.965} C_VEL
LIN {X 0,Y 264.167,Z 415.792,A -85,B 0,C 180,E1 9705.478,E2 9705.478} C_VEL
LIN {X 0,Y 267.41,Z 420.849,A -85,B 0,C 180,E1 9703.044,E2 9703.044} C_VEL
LIN {X 0,Y 272.569,Z 429.455,A -85,B 0,C 180,E1 9699.718,E2 9699.718} C_VEL
LIN {X 0,Y 278.205,Z 439.428,A -85,B 0,C 180,E1 9696.601,E2 9696.601} C_VEL
LIN {X 0,Y 284.489,Z 451.717,A -85,B 0,C 180,E1 9693.547,E2 9693.547} C_VEL
LIN {X 0,Y 287.648,Z 458.573,A -85,B 0,C 180,E1 9692.124,E2 9692.124} C_VEL
LIN {X 0,Y 275.001,Z 617.004,A -85,B 0,C 180,E1 9688.391,E2 9688.391} C_VEL
LIN {X 0,Y 271.734,Z 638.516,A -85,B 0,C 180,E1 9687.623,E2 9687.623} C_VEL
LIN {X 0,Y 267.063,Z 659.339,A -85,B 0,C 180,E1 9686.602,E2 9686.602} C_VEL
LIN {X 0,Y 261.417,Z 678.827,A -85,B 0,C 180,E1 9685.316,E2 9685.316} C_VEL
LIN {X 0,Y 254.677,Z 698.31,A -85,B 0,C 180,E1 9683.591,E2 9683.591} C_VEL
LIN {X 0,Y 247.356,Z 716.687,A -85,B 0,C 180,E1 9681.457,E2 9681.457} C_VEL
LIN {X 0,Y 239.635,Z 734.022,A -85,B 0,C 180,E1 9678.86,E2 9678.86} C_VEL
LIN {X 0,Y 231.751,Z 750.309,A -85,B 0,C 180,E1 9675.739,E2 9675.739} C_VEL
LIN {X 0,Y 224.017,Z 765.478,A -85,B 0,C 180,E1 9672.027,E2 9672.027} C_VEL
LIN {X 0,Y 216.978,Z 779.045,A -85,B 0,C 180,E1 9667.797,E2 9667.797} C_VEL
LIN {X 0,Y 211.224,Z 790.432,A -85,B 0,C 180,E1 9663.304,E2 9663.304} C_VEL
LIN {X 0,Y 206.527,Z 800.636,A -85,B 0,C 180,E1 9658.224,E2 9658.224} C_VEL
LIN {X 0,Y 203.355,Z 809.086,A -85,B 0,C 180,E1 9652.856,E2 9652.856} C_VEL
LIN {X 0,Y 201.67,Z 816.12,A -85,B 0,C 180,E1 9647.008,E2 9647.008} C_VEL
LIN {X 0,Y 201.462,Z 820.977,A -85,B 0,C 180,E1 9641.45,E2 9641.45} C_VEL
LIN {X 0,Y 202.086,Z 823.833,A -85,B 0,C 180,E1 9636.534,E2 9636.534} C_VEL
LIN {X 0,Y 202.75,Z 825.094,A -85,B 0,C 180,E1 9632.261,E2 9632.261} C_VEL
LIN {X 0,Y 202.849,Z 825.217,A -85,B 0,C 180,E1 9628.87,E2 9628.87} C_VEL
LIN {X 0,Y 202.339,Z 824.355,A -85,B 0,C 180,E1 9624.897,E2 9624.897} C_VEL
LIN {X 0,Y 201.598,Z 821.938,A -85,B 0,C 180,E1 9620.004,E2 9620.004} C_VEL
LIN {X 0,Y 201.499,Z 817.583,A -85,B 0,C 180,E1 9614.458,E2 9614.458} C_VEL
LIN {X 0,Y 202.768,Z 811.047,A -85,B 0,C 180,E1 9608.599,E2 9608.599} C_VEL
LIN {X 0,Y 205.767,Z 802.444,A -85,B 0,C 180,E1 9602.822,E2 9602.822} C_VEL
LIN {X 0,Y 210.348,Z 792.203,A -85,B 0,C 180,E1 9597.513,E2 9597.513} C_VEL
LIN {X 0,Y 216.315,Z 780.23,A -85,B 0,C 180,E1 9592.657,E2 9592.657} C_VEL
LIN {X 0,Y 223.133,Z 767.029,A -85,B 0,C 180,E1 9588.445,E2 9588.445} C_VEL
LIN {X 0,Y 230.465,Z 752.665,A -85,B 0,C 180,E1 9584.821,E2 9584.821} C_VEL
LIN {X 0,Y 237.92,Z 737.371,A -85,B 0,C 180,E1 9581.762,E2 9581.762} C_VEL
LIN {X 0,Y 245.336,Z 721.033,A -85,B 0,C 180,E1 9579.175,E2 9579.175} C_VEL
LIN {X 0,Y 252.706,Z 703.05,A -85,B 0,C 180,E1 9576.945,E2 9576.945} C_VEL
LIN {X 0,Y 259.56,Z 683.999,A -85,B 0,C 180,E1 9575.133,E2 9575.133} C_VEL
LIN {X 0,Y 265.618,Z 664.057,A -85,B 0,C 180,E1 9573.708,E2 9573.708} C_VEL
LIN {X 0,Y 270.646,Z 643.104,A -85,B 0,C 180,E1 9572.605,E2 9572.605} C_VEL
LIN {X 0,Y 274.215,Z 621.815,A -85,B 0,C 180,E1 9571.787,E2 9571.787} C_VEL
LIN {X 0,Y 276.809,Z 594.278,A -85,B 0,C 180,E1 9571.056,E2 9571.056} C_VEL
LIN {X 0,Y 287.438,Z 458.04,A -85,B 0,C 180,E1 9567.85,E2 9567.85} C_VEL
LIN {X 0,Y 280.492,Z 443.907,A -85,B 0,C 180,E1 9564.649,E2 9564.649} C_VEL
LIN {X 0,Y 274.522,Z 432.916,A -85,B 0,C 180,E1 9561.527,E2 9561.527} C_VEL
LIN {X 0,Y 269.085,Z 423.759,A -85,B 0,C 180,E1 9558.243,E2 9558.243} C_VEL
LIN {X 0,Y 265.374,Z 417.733,A -85,B 0,C 180,E1 9555.628,E2 9555.628} C_VEL
LIN {X 0,Y 261.94,Z 412.365,A -85,B 0,C 180,E1 9552.79,E2 9552.79} C_VEL
LIN {X 0,Y 259.84,Z 409.19,A -85,B 0,C 180,E1 9550.756,E2 9550.756} C_VEL
LIN {X 0,Y 257.045,Z 404.709,A -85,B 0,C 180,E1 9547.375,E2 9547.375} C_VEL
LIN {X 0,Y 254.133,Z 400.146,A -85,B 0,C 180,E1 9541.803,E2 9541.803} C_VEL
LIN {X 0,Y 253.248,Z 399.042,A -85,B 0,C 180,E1 9535.924,E2 9535.924} C_VEL
LIN {X 0,Y 254.781,Z 400.014,A -85,B 0,C 180,E1 9530.056,E2 9530.056} C_VEL
LIN {X 0,Y 255.635,Z 400.962,A -85,B 0,C 180,E1 9528.379,E2 9528.379} C_VEL
LIN {X 0,Y 259.582,Z 406.049,A -85,B 0,C 180,E1 9523.093,E2 9523.093} C_VEL
LIN {X 0,Y 263.494,Z 411.398,A -85,B 0,C 180,E1 9519.451,E2 9519.451} C_VEL
LIN {X 0,Y 267.138,Z 416.597,A -85,B 0,C 180,E1 9516.683,E2 9516.683} C_VEL
LIN {X 0,Y 270.805,Z 421.953,A -85,B 0,C 180,E1 9514.289,E2 9514.289} C_VEL
LIN {X 0,Y 276.412,Z 430.661,A -85,B 0,C 180,E1 9511.112,E2 9511.112} C_VEL
LIN {X 0,Y 282.804,Z 441.7,A -85,B 0,C 180,E1 9507.972,E2 9507.972} C_VEL
LIN {X 0,Y 287.099,Z 449.953,A -85,B 0,C 180,E1 9506.061,E2 9506.061} C_VEL
LIN {X 0,Y 278.175,Z 576.264,A -85,B 0,C 180,E1 9503.248,E2 9503.248} C_VEL
LIN {X 0,Y 276.24,Z 595.642,A -85,B 0,C 180,E1 9502.549,E2 9502.549} C_VEL
LIN {X 0,Y 273.3,Z 613.874,A -85,B 0,C 180,E1 9501.61,E2 9501.61} C_VEL
LIN {X 0,Y 269.208,Z 632.219,A -85,B 0,C 180,E1 9500.343,E2 9500.343} C_VEL
LIN {X 0,Y 264.064,Z 650.173,A -85,B 0,C 180,E1 9498.728,E2 9498.728} C_VEL
LIN {X 0,Y 258.321,Z 666.619,A -85,B 0,C 180,E1 9496.852,E2 9496.852} C_VEL
LIN {X 0,Y 251.676,Z 682.752,A -85,B 0,C 180,E1 9494.522,E2 9494.522} C_VEL
LIN {X 0,Y 244.577,Z 697.719,A -85,B 0,C 180,E1 9491.785,E2 9491.785} C_VEL
LIN {X 0,Y 237.236,Z 711.482,A -85,B 0,C 180,E1 9488.59,E2 9488.59} C_VEL
LIN {X 0,Y 230.094,Z 723.622,A -85,B 0,C 180,E1 9485,E2 9485} C_VEL
LIN {X 0,Y 223.373,Z 734.214,A -85,B 0,C 180,E1 9480.981,E2 9480.981} C_VEL
LIN {X 0,Y 217.322,Z 743.265,A -85,B 0,C 180,E1 9476.504,E2 9476.504} C_VEL
LIN {X 0,Y 212.138,Z 750.752,A -85,B 0,C 180,E1 9471.569,E2 9471.569} C_VEL
LIN {X 0,Y 208.258,Z 756.378,A -85,B 0,C 180,E1 9466.455,E2 9466.455} C_VEL
LIN {X 0,Y 205.511,Z 760.46,A -85,B 0,C 180,E1 9460.938,E2 9460.938} C_VEL
LIN {X 0,Y 203.998,Z 762.823,A -85,B 0,C 180,E1 9455.343,E2 9455.343} C_VEL
LIN {X 0,Y 203.564,Z 763.564,A -85,B 0,C 180,E1 9449.719,E2 9449.719} C_VEL
LIN {X 0,Y 204.088,Z 762.719,A -85,B 0,C 180,E1 9444.095,E2 9444.095} C_VEL
LIN {X 0,Y 205.702,Z 760.237,A -85,B 0,C 180,E1 9438.505,E2 9438.505} C_VEL
LIN {X 0,Y 208.562,Z 756.013,A -85,B 0,C 180,E1 9432.997,E2 9432.997} C_VEL
LIN {X 0,Y 212.806,Z 749.886,A -85,B 0,C 180,E1 9427.631,E2 9427.631} C_VEL
LIN {X 0,Y 218.173,Z 742.127,A -85,B 0,C 180,E1 9422.724,E2 9422.724} C_VEL
LIN {X 0,Y 224.187,Z 733.116,A -85,B 0,C 180,E1 9418.414,E2 9418.414} C_VEL
LIN {X 0,Y 230.874,Z 722.544,A -85,B 0,C 180,E1 9414.508,E2 9414.508} C_VEL
LIN {X 0,Y 238.068,Z 710.226,A -85,B 0,C 180,E1 9410.953,E2 9410.953} C_VEL
LIN {X 0,Y 245.027,Z 697.109,A -85,B 0,C 180,E1 9407.96,E2 9407.96} C_VEL
LIN {X 0,Y 251.826,Z 682.732,A -85,B 0,C 180,E1 9405.352,E2 9405.352} C_VEL
LIN {X 0,Y 258.482,Z 666.589,A -85,B 0,C 180,E1 9403.024,E2 9403.024} C_VEL
LIN {X 0,Y 264.53,Z 649.256,A -85,B 0,C 180,E1 9401.059,E2 9401.059} C_VEL
LIN {X 0,Y 269.81,Z 630.562,A -85,B 0,C 180,E1 9399.409,E2 9399.409} C_VEL
LIN {X 0,Y 273.95,Z 611.411,A -85,B 0,C 180,E1 9398.129,E2 9398.129} C_VEL
LIN {X 0,Y 276.91,Z 591.815,A -85,B 0,C 180,E1 9397.172,E2 9397.172} C_VEL
LIN {X 0,Y 278.665,Z 571.553,A -85,B 0,C 180,E1 9396.505,E2 9396.505} C_VEL
LIN {X 0,Y 287.196,Z 449.723,A -85,B 0,C 180,E1 9393.791,E2 9393.791} C_VEL
LIN {X 0,Y 281.605,Z 439.42,A -85,B 0,C 180,E1 9391.284,E2 9391.284} C_VEL
LIN {X 0,Y 275.622,Z 429.222,A -85,B 0,C 180,E1 9388.256,E2 9388.256} C_VEL
LIN {X 0,Y 270.553,Z 421.467,A -85,B 0,C 180,E1 9385.326,E2 9385.326} C_VEL
LIN {X 0,Y 265.812,Z 414.52,A -85,B 0,C 180,E1 9382.096,E2 9382.096} C_VEL
LIN {X 0,Y 262.321,Z 409.742,A -85,B 0,C 180,E1 9379.251,E2 9379.251} C_VEL
LIN {X 0,Y 259.022,Z 405.21,A -85,B 0,C 180,E1 9375.907,E2 9375.907} C_VEL
LIN {X 0,Y 255.316,Z 400.383,A -85,B 0,C 180,E1 9370.379,E2 9370.379} C_VEL
LIN {X 0,Y 253.544,Z 399.292,A -85,B 0,C 180,E1 9364.298,E2 9364.298} C_VEL
LIN {X 0,Y 253.773,Z 399.758,A -85,B 0,C 180,E1 9360.41,E2 9360.41} C_VEL
LIN {X 0,Y 254.033,Z 401.002,A -85,B 0,C 180,E1 9358.942,E2 9358.942} C_VEL
LIN {X 0,Y 254.391,Z 405.124,A -85,B 0,C 180,E1 9356.876,E2 9356.876} C_VEL
LIN {X 0,Y 255.3,Z 411.169,A -85,B 0,C 180,E1 9354.154,E2 9354.154} C_VEL
LIN {X 0,Y 256.033,Z 412.675,A -85,B 0,C 180,E1 9352.954,E2 9352.954} C_VEL
LIN {X 0,Y 259.784,Z 418.856,A -85,B 0,C 180,E1 9348.455,E2 9348.455} C_VEL
LIN {X 0,Y 262.574,Z 423.451,A -85,B 0,C 180,E1 9345.895,E2 9345.895} C_VEL
LIN {X 0,Y 265.576,Z 428.32,A -85,B 0,C 180,E1 9343.543,E2 9343.543} C_VEL
LIN {X 0,Y 270.665,Z 437.112,A -85,B 0,C 180,E1 9340.132,E2 9340.132} C_VEL
LIN {X 0,Y 276.337,Z 447.743,A -85,B 0,C 180,E1 9336.885,E2 9336.885} C_VEL
LIN {X 0,Y 282.122,Z 459.501,A -85,B 0,C 180,E1 9333.987,E2 9333.987} C_VEL
LIN {X 0,Y 283.275,Z 462.416,A -85,B 0,C 180,E1 9333.422,E2 9333.422} C_VEL
LIN {X 0,Y 270.604,Z 616.092,A -85,B 0,C 180,E1 9329.809,E2 9329.809} C_VEL
LIN {X 0,Y 267.256,Z 637.577,A -85,B 0,C 180,E1 9329.048,E2 9329.048} C_VEL
LIN {X 0,Y 262.685,Z 657.614,A -85,B 0,C 180,E1 9328.079,E2 9328.079} C_VEL
LIN {X 0,Y 256.869,Z 677.223,A -85,B 0,C 180,E1 9326.81,E2 9326.81} C_VEL
LIN {X 0,Y 250.242,Z 695.894,A -85,B 0,C 180,E1 9325.192,E2 9325.192} C_VEL
LIN {X 0,Y 242.954,Z 713.742,A -85,B 0,C 180,E1 9323.171,E2 9323.171} C_VEL
LIN {X 0,Y 235.181,Z 730.745,A -85,B 0,C 180,E1 9320.691,E2 9320.691} C_VEL
LIN {X 0,Y 227.13,Z 746.833,A -85,B 0,C 180,E1 9317.692,E2 9317.692} C_VEL
LIN {X 0,Y 219.339,Z 761.458,A -85,B 0,C 180,E1 9314.221,E2 9314.221} C_VEL
LIN {X 0,Y 211.672,Z 775.476,A -85,B 0,C 180,E1 9309.97,E2 9309.97} C_VEL
LIN {X 0,Y 204.949,Z 787.885,A -85,B 0,C 180,E1 9305.145,E2 9305.145} C_VEL
LIN {X 0,Y 199.532,Z 798.686,A -85,B 0,C 180,E1 9299.741,E2 9299.741} C_VEL
LIN {X 0,Y 195.73,Z 807.819,A -85,B 0,C 180,E1 9293.8,E2 9293.8} C_VEL
LIN {X 0,Y 193.793,Z 814.866,A -85,B 0,C 180,E1 9287.722,E2 9287.722} C_VEL
LIN {X 0,Y 193.479,Z 819.739,A -85,B 0,C 180,E1 9281.929,E2 9281.929} C_VEL
LIN {X 0,Y 194.102,Z 822.611,A -85,B 0,C 180,E1 9276.804,E2 9276.804} C_VEL
LIN {X 0,Y 194.822,Z 823.889,A -85,B 0,C 180,E1 9272.353,E2 9272.353} C_VEL
LIN {X 0,Y 194.934,Z 824.015,A -85,B 0,C 180,E1 9268.824,E2 9268.824} C_VEL
LIN {X 0,Y 194.421,Z 823.231,A -85,B 0,C 180,E1 9264.985,E2 9264.985} C_VEL
LIN {X 0,Y 193.632,Z 820.899,A -85,B 0,C 180,E1 9259.889,E2 9259.889} C_VEL
LIN {X 0,Y 193.557,Z 816.614,A -85,B 0,C 180,E1 9254.111,E2 9254.111} C_VEL
LIN {X 0,Y 194.953,Z 810.141,A -85,B 0,C 180,E1 9248.014,E2 9248.014} C_VEL
LIN {X 0,Y 197.969,Z 802.088,A -85,B 0,C 180,E1 9242.313,E2 9242.313} C_VEL
LIN {X 0,Y 202.462,Z 792.615,A -85,B 0,C 180,E1 9237.091,E2 9237.091} C_VEL
LIN {X 0,Y 208.492,Z 781.169,A -85,B 0,C 180,E1 9232.133,E2 9232.133} C_VEL
LIN {X 0,Y 215.572,Z 768.227,A -85,B 0,C 180,E1 9227.739,E2 9227.739} C_VEL
LIN {X 0,Y 223.377,Z 753.787,A -85,B 0,C 180,E1 9223.893,E2 9223.893} C_VEL
LIN {X 0,Y 231.624,Z 737.758,A -85,B 0,C 180,E1 9220.56,E2 9220.56} C_VEL
LIN {X 0,Y 239.679,Z 720.833,A -85,B 0,C 180,E1 9217.823,E2 9217.823} C_VEL
LIN {X 0,Y 247.201,Z 703.258,A -85,B 0,C 180,E1 9215.613,E2 9215.613} C_VEL
LIN {X 0,Y 254.038,Z 685.125,A -85,B 0,C 180,E1 9213.856,E2 9213.856} C_VEL
LIN {X 0,Y 260.107,Z 666.247,A -85,B 0,C 180,E1 9212.463,E2 9212.463} C_VEL
LIN {X 0,Y 265.275,Z 646.29,A -85,B 0,C 180,E1 9211.365,E2 9211.365} C_VEL
LIN {X 0,Y 269.18,Z 625.438,A -85,B 0,C 180,E1 9210.515,E2 9210.515} C_VEL
LIN {X 0,Y 271.636,Z 603.776,A -85,B 0,C 180,E1 9209.889,E2 9209.889} C_VEL
LIN {X 0,Y 283.093,Z 461.902,A -85,B 0,C 180,E1 9206.566,E2 9206.566} C_VEL
LIN {X 0,Y 277.185,Z 449.518,A -85,B 0,C 180,E1 9203.659,E2 9203.659} C_VEL
LIN {X 0,Y 271.628,Z 439.041,A -85,B 0,C 180,E1 9200.581,E2 9200.581} C_VEL
LIN {X 0,Y 266.236,Z 429.526,A -85,B 0,C 180,E1 9197.089,E2 9197.089} C_VEL
LIN {X 0,Y 262.995,Z 424.271,A -85,B 0,C 180,E1 9194.644,E2 9194.644} C_VEL
LIN {X 0,Y 260.223,Z 419.713,A -85,B 0,C 180,E1 9192.2,E2 9192.2} C_VEL
LIN {X 0,Y 258.215,Z 416.595,A -85,B 0,C 180,E1 9190.147,E2 9190.147} C_VEL
LIN {X 0,Y 255.73,Z 412.411,A -85,B 0,C 180,E1 9186.961,E2 9186.961} C_VEL
LIN {X 0,Y 253.076,Z 408.03,A -85,B 0,C 180,E1 9181.584,E2 9181.584} C_VEL
LIN {X 0,Y 252.289,Z 406.989,A -85,B 0,C 180,E1 9175.681,E2 9175.681} C_VEL
LIN {X 0,Y 253.926,Z 408.051,A -85,B 0,C 180,E1 9169.793,E2 9169.793} C_VEL
LIN {X 0,Y 254.652,Z 409.134,A -85,B 0,C 180,E1 9168.333,E2 9168.333} C_VEL
LIN {X 0,Y 258.219,Z 413.781,A -85,B 0,C 180,E1 9163.464,E2 9163.464} C_VEL
LIN {X 0,Y 261.959,Z 419.081,A -85,B 0,C 180,E1 9159.85,E2 9159.85} C_VEL
LIN {X 0,Y 265.447,Z 424.21,A -85,B 0,C 180,E1 9157.113,E2 9157.113} C_VEL
LIN {X 0,Y 269.931,Z 430.897,A -85,B 0,C 180,E1 9154.14,E2 9154.14} C_VEL
LIN {X 0,Y 275.966,Z 441,A -85,B 0,C 180,E1 9150.717,E2 9150.717} C_VEL
LIN {X 0,Y 282.464,Z 452.944,A -85,B 0,C 180,E1 9147.539,E2 9147.539} C_VEL
LIN {X 0,Y 282.786,Z 454.006,A -85,B 0,C 180,E1 9147.37,E2 9147.37} C_VEL
LIN {X 0,Y 273.755,Z 577.026,A -85,B 0,C 180,E1 9144.624,E2 9144.624} C_VEL
LIN {X 0,Y 271.752,Z 596.364,A -85,B 0,C 180,E1 9143.925,E2 9143.925} C_VEL
LIN {X 0,Y 268.767,Z 614.358,A -85,B 0,C 180,E1 9143.003,E2 9143.003} C_VEL
LIN {X 0,Y 264.695,Z 632.223,A -85,B 0,C 180,E1 9141.783,E2 9141.783} C_VEL
LIN {X 0,Y 259.577,Z 649.758,A -85,B 0,C 180,E1 9140.23,E2 9140.23} C_VEL
LIN {X 0,Y 253.291,Z 667.268,A -85,B 0,C 180,E1 9138.249,E2 9138.249} C_VEL
LIN {X 0,Y 246.395,Z 683.474,A -85,B 0,C 180,E1 9135.909,E2 9135.909} C_VEL
LIN {X 0,Y 239.01,Z 698.506,A -85,B 0,C 180,E1 9133.154,E2 9133.154} C_VEL
LIN {X 0,Y 231.599,Z 711.922,A -85,B 0,C 180,E1 9130.034,E2 9130.034} C_VEL
LIN {X 0,Y 224.101,Z 724.189,A -85,B 0,C 180,E1 9126.397,E2 9126.397} C_VEL
LIN {X 0,Y 217.005,Z 734.895,A -85,B 0,C 180,E1 9122.307,E2 9122.307} C_VEL
LIN {X 0,Y 210.58,Z 744.05,A -85,B 0,C 180,E1 9117.73,E2 9117.73} C_VEL
LIN {X 0,Y 205.038,Z 751.635,A -85,B 0,C 180,E1 9112.658,E2 9112.658} C_VEL
LIN {X 0,Y 200.85,Z 757.35,A -85,B 0,C 180,E1 9107.378,E2 9107.378} C_VEL
LIN {X 0,Y 197.854,Z 761.519,A -85,B 0,C 180,E1 9101.662,E2 9101.662} C_VEL
LIN {X 0,Y 196.174,Z 763.962,A -85,B 0,C 180,E1 9095.851,E2 9095.851} C_VEL
LIN {X 0,Y 195.656,Z 764.775,A -85,B 0,C 180,E1 9090,E2 9090} C_VEL
LIN {X 0,Y 196.162,Z 763.998,A -85,B 0,C 180,E1 9084.149,E2 9084.149} C_VEL
LIN {X 0,Y 197.823,Z 761.596,A -85,B 0,C 180,E1 9078.336,E2 9078.336} C_VEL
LIN {X 0,Y 200.801,Z 757.468,A -85,B 0,C 180,E1 9072.617,E2 9072.617} C_VEL
LIN {X 0,Y 205.284,Z 751.395,A -85,B 0,C 180,E1 9067.008,E2 9067.008} C_VEL
LIN {X 0,Y 210.828,Z 743.822,A -85,B 0,C 180,E1 9061.998,E2 9061.998} C_VEL
LIN {X 0,Y 217.302,Z 734.606,A -85,B 0,C 180,E1 9057.43,E2 9057.43} C_VEL
LIN {X 0,Y 224.661,Z 723.474,A -85,B 0,C 180,E1 9053.236,E2 9053.236} C_VEL
LIN {X 0,Y 231.984,Z 711.472,A -85,B 0,C 180,E1 9049.719,E2 9049.719} C_VEL
LIN {X 0,Y 239.687,Z 697.456,A -85,B 0,C 180,E1 9046.506,E2 9046.506} C_VEL
LIN {X 0,Y 247.006,Z 682.446,A -85,B 0,C 180,E1 9043.805,E2 9043.805} C_VEL
LIN {X 0,Y 253.758,Z 666.463,A -85,B 0,C 180,E1 9041.529,E2 9041.529} C_VEL
LIN {X 0,Y 259.939,Z 649.121,A -85,B 0,C 180,E1 9039.59,E2 9039.59} C_VEL
LIN {X 0,Y 265.193,Z 630.945,A -85,B 0,C 180,E1 9038.004,E2 9038.004} C_VEL
LIN {X 0,Y 269.4,Z 612.029,A -85,B 0,C 180,E1 9036.746,E2 9036.746} C_VEL
LIN {X 0,Y 272.432,Z 592.635,A -85,B 0,C 180,E1 9035.799,E2 9035.799} C_VEL
LIN {X 0,Y 274.264,Z 572.377,A -85,B 0,C 180,E1 9035.13,E2 9035.13} C_VEL
LIN {X 0,Y 282.882,Z 453.569,A -85,B 0,C 180,E1 9032.467,E2 9032.467} C_VEL
LIN {X 0,Y 276.468,Z 441.753,A -85,B 0,C 180,E1 9029.344,E2 9029.344} C_VEL
LIN {X 0,Y 271.149,Z 432.812,A -85,B 0,C 180,E1 9026.382,E2 9026.382} C_VEL
LIN {X 0,Y 266.347,Z 425.421,A -85,B 0,C 180,E1 9023.273,E2 9023.273} C_VEL
LIN {X 0,Y 263.351,Z 421.042,A -85,B 0,C 180,E1 9021.026,E2 9021.026} C_VEL
LIN {X 0,Y 260.769,Z 417.311,A -85,B 0,C 180,E1 9018.789,E2 9018.789} C_VEL
LIN {X 0,Y 257.678,Z 412.938,A -85,B 0,C 180,E1 9015.53,E2 9015.53} C_VEL
LIN {X 0,Y 254.241,Z 408.276,A -85,B 0,C 180,E1 9010.194,E2 9010.194} C_VEL
LIN {X 0,Y 252.572,Z 407.233,A -85,B 0,C 180,E1 9004.314,E2 9004.314} C_VEL
LIN {X 0,Y 253.333,Z 408.221,A -85,B 0,C 180,E1 8998.417,E2 8998.417} C_VEL
LIN {X 0,Y 256.033,Z 412.675,A -85,B 0,C 180,E1 8992.954,E2 8992.954} C_VEL
LIN {X 0,Y 256.979,Z 414.785,A -85,B 0,C 180,E1 8991.57,E2 8991.57} C_VEL
LIN {X 0,Y 258.033,Z 419.596,A -85,B 0,C 180,E1 8989.915,E2 8989.915} C_VEL
LIN {X 0,Y 259.923,Z 428.541,A -85,B 0,C 180,E1 8987.346,E2 8987.346} C_VEL
LIN {X 0,Y 261.024,Z 431.187,A -85,B 0,C 180,E1 8986.272,E2 8986.272} C_VEL
LIN {X 0,Y 263.962,Z 436.135,A -85,B 0,C 180,E1 8983.892,E2 8983.892} C_VEL
LIN {X 0,Y 268.762,Z 444.869,A -85,B 0,C 180,E1 8980.552,E2 8980.552} C_VEL
LIN {X 0,Y 273.864,Z 454.801,A -85,B 0,C 180,E1 8977.516,E2 8977.516} C_VEL
LIN {X 0,Y 279.077,Z 465.837,A -85,B 0,C 180,E1 8974.772,E2 8974.772} C_VEL
LIN {X 0,Y 266.38,Z 615.165,A -85,B 0,C 180,E1 8971.274,E2 8971.274} C_VEL
LIN {X 0,Y 262.944,Z 636.67,A -85,B 0,C 180,E1 8970.519,E2 8970.519} C_VEL
LIN {X 0,Y 258.07,Z 657.385,A -85,B 0,C 180,E1 8969.523,E2 8969.523} C_VEL
LIN {X 0,Y 252.139,Z 676.761,A -85,B 0,C 180,E1 8968.274,E2 8968.274} C_VEL
LIN {X 0,Y 244.931,Z 696.333,A -85,B 0,C 180,E1 8966.572,E2 8966.572} C_VEL
LIN {X 0,Y 237.126,Z 714.604,A -85,B 0,C 180,E1 8964.466,E2 8964.466} C_VEL
LIN {X 0,Y 228.803,Z 731.913,A -85,B 0,C 180,E1 8961.866,E2 8961.866} C_VEL
LIN {X 0,Y 220.297,Z 748.012,A -85,B 0,C 180,E1 8958.744,E2 8958.744} C_VEL
LIN {X 0,Y 211.941,Z 762.843,A -85,B 0,C 180,E1 8955.042,E2 8955.042} C_VEL
LIN {X 0,Y 204.052,Z 776.444,A -85,B 0,C 180,E1 8950.668,E2 8950.668} C_VEL
LIN {X 0,Y 197.32,Z 788.149,A -85,B 0,C 180,E1 8945.831,E2 8945.831} C_VEL
LIN {X 0,Y 192.074,Z 797.92,A -85,B 0,C 180,E1 8940.673,E2 8940.673} C_VEL
LIN {X 0,Y 188.152,Z 806.55,A -85,B 0,C 180,E1 8934.822,E2 8934.822} C_VEL
LIN {X 0,Y 185.945,Z 813.61,A -85,B 0,C 180,E1 8928.496,E2 8928.496} C_VEL
LIN {X 0,Y 185.499,Z 818.499,A -85,B 0,C 180,E1 8922.451,E2 8922.451} C_VEL
LIN {X 0,Y 186.162,Z 821.531,A -85,B 0,C 180,E1 8916.786,E2 8916.786} C_VEL
LIN {X 0,Y 186.928,Z 822.719,A -85,B 0,C 180,E1 8912.146,E2 8912.146} C_VEL
LIN {X 0,Y 187.015,Z 822.81,A -85,B 0,C 180,E1 8908.759,E2 8908.759} C_VEL
LIN {X 0,Y 186.446,Z 822.014,A -85,B 0,C 180,E1 8904.769,E2 8904.769} C_VEL
LIN {X 0,Y 185.634,Z 819.662,A -85,B 0,C 180,E1 8899.448,E2 8899.448} C_VEL
LIN {X 0,Y 185.656,Z 815.362,A -85,B 0,C 180,E1 8893.416,E2 8893.416} C_VEL
LIN {X 0,Y 187.283,Z 808.876,A -85,B 0,C 180,E1 8887.063,E2 8887.063} C_VEL
LIN {X 0,Y 190.629,Z 800.812,A -85,B 0,C 180,E1 8881.149,E2 8881.149} C_VEL
LIN {X 0,Y 195.495,Z 791.337,A -85,B 0,C 180,E1 8875.766,E2 8875.766} C_VEL
LIN {X 0,Y 201.572,Z 780.562,A -85,B 0,C 180,E1 8870.954,E2 8870.954} C_VEL
LIN {X 0,Y 209.007,Z 767.743,A -85,B 0,C 180,E1 8866.46,E2 8866.46} C_VEL
LIN {X 0,Y 217.161,Z 753.439,A -85,B 0,C 180,E1 8862.553,E2 8862.553} C_VEL
LIN {X 0,Y 225.436,Z 738.145,A -85,B 0,C 180,E1 8859.292,E2 8859.292} C_VEL
LIN {X 0,Y 233.414,Z 722.238,A -85,B 0,C 180,E1 8856.636,E2 8856.636} C_VEL
LIN {X 0,Y 241.151,Z 705.141,A -85,B 0,C 180,E1 8854.404,E2 8854.404} C_VEL
LIN {X 0,Y 248.509,Z 686.643,A -85,B 0,C 180,E1 8852.554,E2 8852.554} C_VEL
LIN {X 0,Y 255.094,Z 667.118,A -85,B 0,C 180,E1 8851.085,E2 8851.085} C_VEL
LIN {X 0,Y 260.539,Z 647.028,A -85,B 0,C 180,E1 8849.966,E2 8849.966} C_VEL
LIN {X 0,Y 264.728,Z 625.774,A -85,B 0,C 180,E1 8849.09,E2 8849.09} C_VEL
LIN {X 0,Y 267.336,Z 604.079,A -85,B 0,C 180,E1 8848.456,E2 8848.456} C_VEL
